LIN {X 0,Y 547.495,Z 446.55,A -85,B 0,C 180,E1 25697.348,E2 25697.348} C_VEL
LIN {X 0,Y 546.646,Z 474.266,A -85,B 0,C 180,E1 25694.031,E2 25694.031} C_VEL
LIN {X 0,Y 545.935,Z 503.573,A -85,B 0,C 180,E1 25690.623,E2 25690.623} C_VEL
LIN {X 0,Y 545.225,Z 533.992,A -85,B 0,C 180,E1 25687.109,E2 25687.109} C_VEL
LIN {X 0,Y 544.841,Z 556.823,A -85,B 0,C 180,E1 25684.577,E2 25684.577} C_VEL
LIN {X 0,Y 545.708,Z 565.508,A -85,B 0,C 180,E1 25684.415,E2 25684.415} C_VEL
LIN {X 0,Y 545.328,Z 668.465,A -85,B 0,C 180,E1 25683.029,E2 25683.029} C_VEL
LIN {X 0,Y 545.205,Z 683.51,A -85,B 0,C 180,E1 25682.627,E2 25682.627} C_VEL
LIN {X 0,Y 545.001,Z 698.163,A -85,B 0,C 180,E1 25682.019,E2 25682.019} C_VEL
LIN {X 0,Y 544.742,Z 711.794,A -85,B 0,C 180,E1 25681.233,E2 25681.233} C_VEL
LIN {X 0,Y 544.518,Z 723.816,A -85,B 0,C 180,E1 25680.329,E2 25680.329} C_VEL
LIN {X 0,Y 544.318,Z 735.754,A -85,B 0,C 180,E1 25679.174,E2 25679.174} C_VEL
LIN {X 0,Y 544.144,Z 746.013,A -85,B 0,C 180,E1 25677.891,E2 25677.891} C_VEL
LIN {X 0,Y 544.028,Z 754.441,A -85,B 0,C 180,E1 25676.526,E2 25676.526} C_VEL
LIN {X 0,Y 543.96,Z 761.021,A -85,B 0,C 180,E1 25675.125,E2 25675.125} C_VEL
LIN {X 0,Y 543.928,Z 766.386,A -85,B 0,C 180,E1 25673.509,E2 25673.509} C_VEL
LIN {X 0,Y 543.917,Z 769.602,A -85,B 0,C 180,E1 25671.911,E2 25671.911} C_VEL
LIN {X 0,Y 543.918,Z 770.918,A -85,B 0,C 180,E1 25670.362,E2 25670.362} C_VEL
LIN {X 0,Y 543.916,Z 770.49,A -85,B 0,C 180,E1 25668.765,E2 25668.765} C_VEL
LIN {X 0,Y 543.919,Z 768.037,A -85,B 0,C 180,E1 25667.105,E2 25667.105} C_VEL
LIN {X 0,Y 543.939,Z 763.873,A -85,B 0,C 180,E1 25665.567,E2 25665.567} C_VEL
LIN {X 0,Y 543.985,Z 758.294,A -85,B 0,C 180,E1 25664.15,E2 25664.15} C_VEL
LIN {X 0,Y 544.074,Z 750.741,A -85,B 0,C 180,E1 25662.74,E2 25662.74} C_VEL
LIN {X 0,Y 544.199,Z 742.577,A -85,B 0,C 180,E1 25661.552,E2 25661.552} C_VEL
LIN {X 0,Y 544.392,Z 731.756,A -85,B 0,C 180,E1 25660.316,E2 25660.316} C_VEL
LIN {X 0,Y 544.604,Z 719.668,A -85,B 0,C 180,E1 25659.244,E2 25659.244} C_VEL
LIN {X 0,Y 544.841,Z 707.24,A -85,B 0,C 180,E1 25658.389,E2 25658.389} C_VEL
LIN {X 0,Y 545.065,Z 694.016,A -85,B 0,C 180,E1 25657.695,E2 25657.695} C_VEL
LIN {X 0,Y 545.26,Z 679.155,A -85,B 0,C 180,E1 25657.146,E2 25657.146} C_VEL
LIN {X 0,Y 545.39,Z 664.539,A -85,B 0,C 180,E1 25656.811,E2 25656.811} C_VEL
LIN {X 0,Y 545.478,Z 561.409,A -85,B 0,C 180,E1 25655.434,E2 25655.434} C_VEL
LIN {X 0,Y 544.883,Z 556.572,A -85,B 0,C 180,E1 25655.317,E2 25655.317} C_VEL
LIN {X 0,Y 545.301,Z 528.031,A -85,B 0,C 180,E1 25652.122,E2 25652.122} C_VEL
LIN {X 0,Y 546.018,Z 497.792,A -85,B 0,C 180,E1 25648.636,E2 25648.636} C_VEL
LIN {X 0,Y 546.669,Z 469.731,A -85,B 0,C 180,E1 25645.384,E2 25645.384} C_VEL
LIN {X 0,Y 547.326,Z 446.384,A -85,B 0,C 180,E1 25642.6,E2 25642.6} C_VEL
LIN {X 0,Y 544.355,Z 435.109,A -85,B 0,C 180,E1 25640.991,E2 25640.991} C_VEL
LIN {X 0,Y 544.39,Z 434.987,A -85,B 0,C 180,E1 25637.806,E2 25637.806} C_VEL
LIN {X 0,Y 544.328,Z 434.99,A -85,B 0,C 180,E1 25634.553,E2 25634.553} C_VEL
LIN {X 0,Y 544.383,Z 434.988,A -85,B 0,C 180,E1 25631.362,E2 25631.362} C_VEL
LIN {X 0,Y 544.329,Z 434.988,A -85,B 0,C 180,E1 25628.22,E2 25628.22} C_VEL
LIN {X 0,Y 544.332,Z 434.989,A -85,B 0,C 180,E1 25624.776,E2 25624.776} C_VEL
LIN {X 0,Y 544.365,Z 434.988,A -85,B 0,C 180,E1 25621.619,E2 25621.619} C_VEL
LIN {X 0,Y 544.318,Z 434.988,A -85,B 0,C 180,E1 25618.431,E2 25618.431} C_VEL
LIN {X 0,Y 544.386,Z 434.991,A -85,B 0,C 180,E1 25615.294,E2 25615.294} C_VEL
LIN {X 0,Y 544.32,Z 434.987,A -85,B 0,C 180,E1 25612.155,E2 25612.155} C_VEL
LIN {X 0,Y 544.373,Z 434.983,A -85,B 0,C 180,E1 25608.887,E2 25608.887} C_VEL
LIN {X 0,Y 544.336,Z 434.987,A -85,B 0,C 180,E1 25605.733,E2 25605.733} C_VEL
LIN {X 0,Y 544.34,Z 434.982,A -85,B 0,C 180,E1 25602.386,E2 25602.386} C_VEL
LIN {X 0,Y 544.365,Z 434.986,A -85,B 0,C 180,E1 25599.322,E2 25599.322} C_VEL
LIN {X 0,Y 544.333,Z 434.985,A -85,B 0,C 180,E1 25596.001,E2 25596.001} C_VEL
LIN {X 0,Y 544.4,Z 434.984,A -85,B 0,C 180,E1 25592.735,E2 25592.735} C_VEL
LIN {X 0,Y 544.34,Z 434.987,A -85,B 0,C 180,E1 25589.611,E2 25589.611} C_VEL
LIN {X 0,Y 544.365,Z 434.976,A -85,B 0,C 180,E1 25586.274,E2 25586.274} C_VEL
LIN {X 0,Y 544.375,Z 434.986,A -85,B 0,C 180,E1 25583.031,E2 25583.031} C_VEL
LIN {X 0,Y 544.346,Z 434.983,A -85,B 0,C 180,E1 25579.754,E2 25579.754} C_VEL
LIN {X 0,Y 544.404,Z 434.98,A -85,B 0,C 180,E1 25576.43,E2 25576.43} C_VEL
LIN {X 0,Y 544.357,Z 434.987,A -85,B 0,C 180,E1 25573.165,E2 25573.165} C_VEL
LIN {X 0,Y 544.359,Z 434.976,A -85,B 0,C 180,E1 25569.729,E2 25569.729} C_VEL
LIN {X 0,Y 544.405,Z 434.985,A -85,B 0,C 180,E1 25566.433,E2 25566.433} C_VEL
LIN {X 0,Y 544.356,Z 434.985,A -85,B 0,C 180,E1 25563.159,E2 25563.159} C_VEL
LIN {X 0,Y 544.382,Z 434.974,A -85,B 0,C 180,E1 25559.79,E2 25559.79} C_VEL
LIN {X 0,Y 544.399,Z 434.989,A -85,B 0,C 180,E1 25556.42,E2 25556.42} C_VEL
LIN {X 0,Y 544.36,Z 434.98,A -85,B 0,C 180,E1 25553.143,E2 25553.143} C_VEL
LIN {X 0,Y 544.402,Z 434.981,A -85,B 0,C 180,E1 25549.845,E2 25549.845} C_VEL
LIN {X 0,Y 544.385,Z 434.987,A -85,B 0,C 180,E1 25546.511,E2 25546.511} C_VEL
LIN {X 0,Y 544.37,Z 434.981,A -85,B 0,C 180,E1 25543.125,E2 25543.125} C_VEL
LIN {X 0,Y 544.401,Z 434.979,A -85,B 0,C 180,E1 25539.801,E2 25539.801} C_VEL
LIN {X 0,Y 544.383,Z 434.985,A -85,B 0,C 180,E1 25536.421,E2 25536.421} C_VEL
LIN {X 0,Y 544.376,Z 434.977,A -85,B 0,C 180,E1 25532.975,E2 25532.975} C_VEL
LIN {X 0,Y 544.4,Z 434.981,A -85,B 0,C 180,E1 25529.664,E2 25529.664} C_VEL
LIN {X 0,Y 544.385,Z 434.986,A -85,B 0,C 180,E1 25526.307,E2 25526.307} C_VEL
LIN {X 0,Y 544.382,Z 434.982,A -85,B 0,C 180,E1 25522.824,E2 25522.824} C_VEL
LIN {X 0,Y 544.396,Z 434.984,A -85,B 0,C 180,E1 25519.446,E2 25519.446} C_VEL
LIN {X 0,Y 544.394,Z 434.988,A -85,B 0,C 180,E1 25516.032,E2 25516.032} C_VEL
LIN {X 0,Y 544.384,Z 434.983,A -85,B 0,C 180,E1 25512.565,E2 25512.565} C_VEL
LIN {X 0,Y 544.393,Z 434.986,A -85,B 0,C 180,E1 25509.32,E2 25509.32} C_VEL
LIN {X 0,Y 544.389,Z 434.986,A -85,B 0,C 180,E1 25505.996,E2 25505.996} C_VEL
LIN {X 0,Y 544.429,Z 435.199,A -85,B 0,C 180,E1 25502.883,E2 25502.883} C_VEL
LIN {X 0,Y 549.545,Z 450.788,A -85,B 0,C 180,E1 25501.295,E2 25501.295} C_VEL
LIN {X 0,Y 548.617,Z 495.169,A -85,B 0,C 180,E1 25498.048,E2 25498.048} C_VEL
LIN {X 0,Y 547.868,Z 539.196,A -85,B 0,C 180,E1 25494.93,E2 25494.93} C_VEL
LIN {X 0,Y 549.12,Z 548.98,A -85,B 0,C 180,E1 25494.728,E2 25494.728} C_VEL
LIN {X 0,Y 548,Z 748.309,A -85,B 0,C 180,E1 25491.965,E2 25491.965} C_VEL
LIN {X 0,Y 547.672,Z 767.397,A -85,B 0,C 180,E1 25491.502,E2 25491.502} C_VEL
LIN {X 0,Y 547.282,Z 785.391,A -85,B 0,C 180,E1 25490.871,E2 25490.871} C_VEL
LIN {X 0,Y 546.836,Z 803.036,A -85,B 0,C 180,E1 25490.05,E2 25490.05} C_VEL
LIN {X 0,Y 546.334,Z 819.765,A -85,B 0,C 180,E1 25489.067,E2 25489.067} C_VEL
LIN {X 0,Y 545.853,Z 835.621,A -85,B 0,C 180,E1 25487.923,E2 25487.923} C_VEL
LIN {X 0,Y 545.378,Z 850.553,A -85,B 0,C 180,E1 25486.619,E2 25486.619} C_VEL
LIN {X 0,Y 544.96,Z 864.211,A -85,B 0,C 180,E1 25485.188,E2 25485.188} C_VEL
LIN {X 0,Y 544.601,Z 876.913,A -85,B 0,C 180,E1 25483.592,E2 25483.592} C_VEL
LIN {X 0,Y 544.329,Z 888.228,A -85,B 0,C 180,E1 25481.872,E2 25481.872} C_VEL
LIN {X 0,Y 544.13,Z 897.993,A -85,B 0,C 180,E1 25480.054,E2 25480.054} C_VEL
LIN {X 0,Y 544.008,Z 906.176,A -85,B 0,C 180,E1 25478.136,E2 25478.136} C_VEL
LIN {X 0,Y 543.945,Z 912.412,A -85,B 0,C 180,E1 25476.226,E2 25476.226} C_VEL
LIN {X 0,Y 543.921,Z 916.878,A -85,B 0,C 180,E1 25474.323,E2 25474.323} C_VEL
LIN {X 0,Y 543.914,Z 919.793,A -85,B 0,C 180,E1 25472.318,E2 25472.318} C_VEL
LIN {X 0,Y 543.908,Z 920.94,A -85,B 0,C 180,E1 25470.316,E2 25470.316} C_VEL
LIN {X 0,Y 543.913,Z 920.347,A -85,B 0,C 180,E1 25468.315,E2 25468.315} C_VEL
LIN {X 0,Y 543.915,Z 918.002,A -85,B 0,C 180,E1 25466.311,E2 25466.311} C_VEL
LIN {X 0,Y 543.931,Z 914.097,A -85,B 0,C 180,E1 25464.409,E2 25464.409} C_VEL
LIN {X 0,Y 543.981,Z 908.468,A -85,B 0,C 180,E1 25462.502,E2 25462.502} C_VEL
LIN {X 0,Y 544.074,Z 901.428,A -85,B 0,C 180,E1 25460.693,E2 25460.693} C_VEL
LIN {X 0,Y 544.234,Z 892.518,A -85,B 0,C 180,E1 25458.878,E2 25458.878} C_VEL
LIN {X 0,Y 544.472,Z 882.154,A -85,B 0,C 180,E1 25457.162,E2 25457.162} C_VEL
LIN {X 0,Y 544.779,Z 870.352,A -85,B 0,C 180,E1 25455.546,E2 25455.546} C_VEL
LIN {X 0,Y 545.178,Z 857.081,A -85,B 0,C 180,E1 25454.032,E2 25454.032} C_VEL
LIN {X 0,Y 545.65,Z 842.222,A -85,B 0,C 180,E1 25452.622,E2 25452.622} C_VEL
LIN {X 0,Y 546.157,Z 826.235,A -85,B 0,C 180,E1 25451.37,E2 25451.37} C_VEL
LIN {X 0,Y 546.65,Z 809.054,A -85,B 0,C 180,E1 25450.278,E2 25450.278} C_VEL
LIN {X 0,Y 547.127,Z 791.811,A -85,B 0,C 180,E1 25449.403,E2 25449.403} C_VEL
LIN {X 0,Y 547.538,Z 773.536,A -85,B 0,C 180,E1 25448.691,E2 25448.691} C_VEL
LIN {X 0,Y 547.894,Z 754.924,A -85,B 0,C 180,E1 25448.174,E2 25448.174} C_VEL
LIN {X 0,Y 548.116,Z 734.498,A -85,B 0,C 180,E1 25447.82,E2 25447.82} C_VEL
LIN {X 0,Y 548.952,Z 546.145,A -85,B 0,C 180,E1 25445.224,E2 25445.224} C_VEL
LIN {X 0,Y 547.799,Z 538.331,A -85,B 0,C 180,E1 25445.034,E2 25445.034} C_VEL
LIN {X 0,Y 548.663,Z 492.747,A -85,B 0,C 180,E1 25441.777,E2 25441.777} C_VEL
LIN {X 0,Y 549.55,Z 450.377,A -85,B 0,C 180,E1 25438.675,E2 25438.675} C_VEL
LIN {X 0,Y 544.437,Z 435.251,A -85,B 0,C 180,E1 25437.134,E2 25437.134} C_VEL
LIN {X 0,Y 544.389,Z 434.988,A -85,B 0,C 180,E1 25433.874,E2 25433.874} C_VEL
LIN {X 0,Y 544.392,Z 434.986,A -85,B 0,C 180,E1 25430.479,E2 25430.479} C_VEL
LIN {X 0,Y 544.4,Z 434.978,A -85,B 0,C 180,E1 25427.048,E2 25427.048} C_VEL
LIN {X 0,Y 544.388,Z 434.986,A -85,B 0,C 180,E1 25423.644,E2 25423.644} C_VEL
LIN {X 0,Y 544.394,Z 434.986,A -85,B 0,C 180,E1 25420.278,E2 25420.278} C_VEL
LIN {X 0,Y 544.4,Z 434.98,A -85,B 0,C 180,E1 25416.911,E2 25416.911} C_VEL
LIN {X 0,Y 544.386,Z 434.984,A -85,B 0,C 180,E1 25413.436,E2 25413.436} C_VEL
LIN {X 0,Y 544.393,Z 434.985,A -85,B 0,C 180,E1 25410.093,E2 25410.093} C_VEL
LIN {X 0,Y 544.395,Z 434.98,A -85,B 0,C 180,E1 25406.742,E2 25406.742} C_VEL
LIN {X 0,Y 544.387,Z 434.985,A -85,B 0,C 180,E1 25403.259,E2 25403.259} C_VEL
LIN {X 0,Y 544.394,Z 434.984,A -85,B 0,C 180,E1 25399.888,E2 25399.888} C_VEL
LIN {X 0,Y 544.4,Z 434.979,A -85,B 0,C 180,E1 25396.43,E2 25396.43} C_VEL
LIN {X 0,Y 544.385,Z 434.986,A -85,B 0,C 180,E1 25393.056,E2 25393.056} C_VEL
LIN {X 0,Y 544.393,Z 434.981,A -85,B 0,C 180,E1 25389.728,E2 25389.728} C_VEL
LIN {X 0,Y 544.393,Z 434.98,A -85,B 0,C 180,E1 25386.327,E2 25386.327} C_VEL
LIN {X 0,Y 544.384,Z 434.986,A -85,B 0,C 180,E1 25382.842,E2 25382.842} C_VEL
LIN {X 0,Y 544.395,Z 434.98,A -85,B 0,C 180,E1 25379.474,E2 25379.474} C_VEL
LIN {X 0,Y 544.392,Z 434.979,A -85,B 0,C 180,E1 25376.103,E2 25376.103} C_VEL
LIN {X 0,Y 544.385,Z 434.986,A -85,B 0,C 180,E1 25372.659,E2 25372.659} C_VEL
LIN {X 0,Y 544.395,Z 434.98,A -85,B 0,C 180,E1 25369.296,E2 25369.296} C_VEL
LIN {X 0,Y 544.393,Z 434.977,A -85,B 0,C 180,E1 25365.871,E2 25365.871} C_VEL
LIN {X 0,Y 544.381,Z 434.984,A -85,B 0,C 180,E1 25362.409,E2 25362.409} C_VEL
LIN {X 0,Y 544.397,Z 434.985,A -85,B 0,C 180,E1 25359.013,E2 25359.013} C_VEL
LIN {X 0,Y 544.395,Z 434.977,A -85,B 0,C 180,E1 25355.591,E2 25355.591} C_VEL
LIN {X 0,Y 544.382,Z 434.987,A -85,B 0,C 180,E1 25352.191,E2 25352.191} C_VEL
LIN {X 0,Y 544.4,Z 434.982,A -85,B 0,C 180,E1 25349.102,E2 25349.102} C_VEL
LIN {X 0,Y 543.39,Z 435.113,A -85,B 0,C 180,E1 25348.291,E2 25348.291} C_VEL
LIN {X 0,Y 536.961,Z 435.911,A -85,B 0,C 180,E1 25346.014,E2 25346.014} C_VEL
LIN {X 0,Y 536.452,Z 435.971,A -85,B 0,C 180,E1 25345.421,E2 25345.421} C_VEL
LIN {X 0,Y 536.445,Z 435.977,A -85,B 0,C 180,E1 25342.037,E2 25342.037} C_VEL
LIN {X 0,Y 536.485,Z 436.227,A -85,B 0,C 180,E1 25339.335,E2 25339.335} C_VEL
LIN {X 0,Y 539.968,Z 449.754,A -85,B 0,C 180,E1 25337.406,E2 25337.406} C_VEL
LIN {X 0,Y 538.979,Z 478.583,A -85,B 0,C 180,E1 25333.932,E2 25333.932} C_VEL
LIN {X 0,Y 538.235,Z 506.906,A -85,B 0,C 180,E1 25330.6,E2 25330.6} C_VEL
LIN {X 0,Y 537.432,Z 537.08,A -85,B 0,C 180,E1 25327.069,E2 25327.069} C_VEL
LIN {X 0,Y 537.047,Z 556.841,A -85,B 0,C 180,E1 25324.835,E2 25324.835} C_VEL
LIN {X 0,Y 538.032,Z 566.096,A -85,B 0,C 180,E1 25324.647,E2 25324.647} C_VEL
LIN {X 0,Y 537.537,Z 668.696,A -85,B 0,C 180,E1 25323.219,E2 25323.219} C_VEL
LIN {X 0,Y 537.393,Z 683.257,A -85,B 0,C 180,E1 25322.823,E2 25322.823} C_VEL
LIN {X 0,Y 537.162,Z 698.051,A -85,B 0,C 180,E1 25322.203,E2 25322.203} C_VEL
LIN {X 0,Y 536.879,Z 711.35,A -85,B 0,C 180,E1 25321.43,E2 25321.43} C_VEL
LIN {X 0,Y 536.617,Z 723.478,A -85,B 0,C 180,E1 25320.513,E2 25320.513} C_VEL
LIN {X 0,Y 536.389,Z 735.343,A -85,B 0,C 180,E1 25319.357,E2 25319.357} C_VEL
LIN {X 0,Y 536.194,Z 745.279,A -85,B 0,C 180,E1 25318.112,E2 25318.112} C_VEL
LIN {X 0,Y 536.062,Z 753.333,A -85,B 0,C 180,E1 25316.832,E2 25316.832} C_VEL
LIN {X 0,Y 535.971,Z 760.681,A -85,B 0,C 180,E1 25315.29,E2 25315.29} C_VEL
LIN {X 0,Y 535.932,Z 765.819,A -85,B 0,C 180,E1 25313.764,E2 25313.764} C_VEL
LIN {X 0,Y 535.919,Z 769.129,A -85,B 0,C 180,E1 25312.255,E2 25312.255} C_VEL
LIN {X 0,Y 535.918,Z 770.822,A -85,B 0,C 180,E1 25310.647,E2 25310.647} C_VEL
LIN {X 0,Y 535.916,Z 770.693,A -85,B 0,C 180,E1 25309.056,E2 25309.056} C_VEL
LIN {X 0,Y 535.919,Z 768.842,A -85,B 0,C 180,E1 25307.48,E2 25307.48} C_VEL
LIN {X 0,Y 535.937,Z 764.857,A -85,B 0,C 180,E1 25305.806,E2 25305.806} C_VEL
LIN {X 0,Y 535.987,Z 759.124,A -85,B 0,C 180,E1 25304.255,E2 25304.255} C_VEL
LIN {X 0,Y 536.082,Z 751.872,A -85,B 0,C 180,E1 25302.823,E2 25302.823} C_VEL
LIN {X 0,Y 536.233,Z 743.203,A -85,B 0,C 180,E1 25301.508,E2 25301.508} C_VEL
LIN {X 0,Y 536.453,Z 732.279,A -85,B 0,C 180,E1 25300.227,E2 25300.227} C_VEL
LIN {X 0,Y 536.689,Z 720.664,A -85,B 0,C 180,E1 25299.165,E2 25299.165} C_VEL
LIN {X 0,Y 536.953,Z 708.57,A -85,B 0,C 180,E1 25298.297,E2 25298.297} C_VEL
LIN {X 0,Y 537.22,Z 694.554,A -85,B 0,C 180,E1 25297.539,E2 25297.539} C_VEL
LIN {X 0,Y 537.436,Z 680.185,A -85,B 0,C 180,E1 25296.989,E2 25296.989} C_VEL
LIN {X 0,Y 537.598,Z 665.309,A -85,B 0,C 180,E1 25296.628,E2 25296.628} C_VEL
LIN {X 0,Y 537.808,Z 562.279,A -85,B 0,C 180,E1 25295.207,E2 25295.207} C_VEL
LIN {X 0,Y 537.071,Z 556.649,A -85,B 0,C 180,E1 25295.073,E2 25295.073} C_VEL
LIN {X 0,Y 537.587,Z 528.08,A -85,B 0,C 180,E1 25291.812,E2 25291.812} C_VEL
LIN {X 0,Y 538.382,Z 497.987,A -85,B 0,C 180,E1 25288.297,E2 25288.297} C_VEL
LIN {X 0,Y 539.146,Z 469.958,A -85,B 0,C 180,E1 25284.999,E2 25284.999} C_VEL
LIN {X 0,Y 539.763,Z 448.718,A -85,B 0,C 180,E1 25282.442,E2 25282.442} C_VEL
LIN {X 0,Y 536.412,Z 436.103,A -85,B 0,C 180,E1 25280.613,E2 25280.613} C_VEL
LIN {X 0,Y 536.428,Z 435.978,A -85,B 0,C 180,E1 25277.294,E2 25277.294} C_VEL
LIN {X 0,Y 536.402,Z 435.978,A -85,B 0,C 180,E1 25274.208,E2 25274.208} C_VEL
LIN {X 0,Y 536.391,Z 435.977,A -85,B 0,C 180,E1 25270.735,E2 25270.735} C_VEL
LIN {X 0,Y 536.455,Z 435.965,A -85,B 0,C 180,E1 25267.537,E2 25267.537} C_VEL
LIN {X 0,Y 536.384,Z 435.978,A -85,B 0,C 180,E1 25264.257,E2 25264.257} C_VEL
LIN {X 0,Y 536.404,Z 435.979,A -85,B 0,C 180,E1 25260.889,E2 25260.889} C_VEL
LIN {X 0,Y 536.399,Z 435.976,A -85,B 0,C 180,E1 25257.784,E2 25257.784} C_VEL
LIN {X 0,Y 536.384,Z 435.977,A -85,B 0,C 180,E1 25254.437,E2 25254.437} C_VEL
LIN {X 0,Y 536.456,Z 435.977,A -85,B 0,C 180,E1 25251.177,E2 25251.177} C_VEL
LIN {X 0,Y 536.387,Z 435.973,A -85,B 0,C 180,E1 25247.994,E2 25247.994} C_VEL
LIN {X 0,Y 536.419,Z 435.976,A -85,B 0,C 180,E1 25244.645,E2 25244.645} C_VEL
LIN {X 0,Y 536.413,Z 435.972,A -85,B 0,C 180,E1 25241.468,E2 25241.468} C_VEL
LIN {X 0,Y 536.395,Z 435.977,A -85,B 0,C 180,E1 25238.097,E2 25238.097} C_VEL
LIN {X 0,Y 536.458,Z 435.966,A -85,B 0,C 180,E1 25234.904,E2 25234.904} C_VEL
LIN {X 0,Y 536.399,Z 435.975,A -85,B 0,C 180,E1 25231.713,E2 25231.713} C_VEL
LIN {X 0,Y 536.432,Z 435.97,A -85,B 0,C 180,E1 25228.379,E2 25228.379} C_VEL
LIN {X 0,Y 536.426,Z 435.967,A -85,B 0,C 180,E1 25225.149,E2 25225.149} C_VEL
LIN {X 0,Y 536.407,Z 435.975,A -85,B 0,C 180,E1 25221.774,E2 25221.774} C_VEL
LIN {X 0,Y 536.461,Z 435.961,A -85,B 0,C 180,E1 25218.473,E2 25218.473} C_VEL
LIN {X 0,Y 536.414,Z 435.972,A -85,B 0,C 180,E1 25215.238,E2 25215.238} C_VEL
LIN {X 0,Y 536.417,Z 435.972,A -85,B 0,C 180,E1 25211.723,E2 25211.723} C_VEL
LIN {X 0,Y 536.465,Z 435.964,A -85,B 0,C 180,E1 25208.467,E2 25208.467} C_VEL
LIN {X 0,Y 536.419,Z 435.974,A -85,B 0,C 180,E1 25205.133,E2 25205.133} C_VEL
LIN {X 0,Y 536.432,Z 435.966,A -85,B 0,C 180,E1 25201.709,E2 25201.709} C_VEL
LIN {X 0,Y 536.465,Z 435.97,A -85,B 0,C 180,E1 25198.398,E2 25198.398} C_VEL
LIN {X 0,Y 536.421,Z 435.974,A -85,B 0,C 180,E1 25195.082,E2 25195.082} C_VEL
LIN {X 0,Y 536.457,Z 435.963,A -85,B 0,C 180,E1 25191.749,E2 25191.749} C_VEL
LIN {X 0,Y 536.457,Z 435.977,A -85,B 0,C 180,E1 25188.388,E2 25188.388} C_VEL
LIN {X 0,Y 536.425,Z 435.966,A -85,B 0,C 180,E1 25184.984,E2 25184.984} C_VEL
LIN {X 0,Y 536.462,Z 435.97,A -85,B 0,C 180,E1 25181.64,E2 25181.64} C_VEL
LIN {X 0,Y 536.463,Z 435.97,A -85,B 0,C 180,E1 25178.152,E2 25178.152} C_VEL
LIN {X 0,Y 536.434,Z 435.973,A -85,B 0,C 180,E1 25174.733,E2 25174.733} C_VEL
LIN {X 0,Y 536.467,Z 435.969,A -85,B 0,C 180,E1 25171.381,E2 25171.381} C_VEL
LIN {X 0,Y 536.464,Z 435.972,A -85,B 0,C 180,E1 25167.915,E2 25167.915} C_VEL
LIN {X 0,Y 536.438,Z 435.972,A -85,B 0,C 180,E1 25164.54,E2 25164.54} C_VEL
LIN {X 0,Y 536.462,Z 435.967,A -85,B 0,C 180,E1 25161.09,E2 25161.09} C_VEL
LIN {X 0,Y 536.461,Z 435.973,A -85,B 0,C 180,E1 25157.714,E2 25157.714} C_VEL
LIN {X 0,Y 536.444,Z 435.972,A -85,B 0,C 180,E1 25154.298,E2 25154.298} C_VEL
LIN {X 0,Y 536.463,Z 435.971,A -85,B 0,C 180,E1 25150.826,E2 25150.826} C_VEL
LIN {X 0,Y 536.456,Z 435.977,A -85,B 0,C 180,E1 25147.417,E2 25147.417} C_VEL
LIN {X 0,Y 536.451,Z 435.976,A -85,B 0,C 180,E1 25143.997,E2 25143.997} C_VEL
LIN {X 0,Y 536.508,Z 436.346,A -85,B 0,C 180,E1 25143.282,E2 25143.282} C_VEL
LIN {X 0,Y 542.232,Z 453.381,A -85,B 0,C 180,E1 25141.524,E2 25141.524} C_VEL
LIN {X 0,Y 541.159,Z 496.053,A -85,B 0,C 180,E1 25138.349,E2 25138.349} C_VEL
LIN {X 0,Y 540.28,Z 539.241,A -85,B 0,C 180,E1 25135.245,E2 25135.245} C_VEL
LIN {X 0,Y 541.72,Z 550.007,A -85,B 0,C 180,E1 25135.037,E2 25135.037} C_VEL
LIN {X 0,Y 540.616,Z 745.193,A -85,B 0,C 180,E1 25132.336,E2 25132.336} C_VEL
LIN {X 0,Y 540.277,Z 763.946,A -85,B 0,C 180,E1 25131.913,E2 25131.913} C_VEL
LIN {X 0,Y 539.846,Z 781.952,A -85,B 0,C 180,E1 25131.312,E2 25131.312} C_VEL
LIN {X 0,Y 539.37,Z 799.844,A -85,B 0,C 180,E1 25130.51,E2 25130.51} C_VEL
LIN {X 0,Y 538.786,Z 817.24,A -85,B 0,C 180,E1 25129.514,E2 25129.514} C_VEL
LIN {X 0,Y 538.22,Z 833.955,A -85,B 0,C 180,E1 25128.324,E2 25128.324} C_VEL
LIN {X 0,Y 537.655,Z 849.441,A -85,B 0,C 180,E1 25126.976,E2 25126.976} C_VEL
LIN {X 0,Y 537.171,Z 863.091,A -85,B 0,C 180,E1 25125.547,E2 25125.547} C_VEL
LIN {X 0,Y 536.736,Z 876.14,A -85,B 0,C 180,E1 25123.905,E2 25123.905} C_VEL
LIN {X 0,Y 536.408,Z 887.592,A -85,B 0,C 180,E1 25122.16,E2 25122.16} C_VEL
LIN {X 0,Y 536.175,Z 897.478,A -85,B 0,C 180,E1 25120.313,E2 25120.313} C_VEL
LIN {X 0,Y 536.036,Z 905.771,A -85,B 0,C 180,E1 25118.366,E2 25118.366} C_VEL
LIN {X 0,Y 535.953,Z 912.109,A -85,B 0,C 180,E1 25116.427,E2 25116.427} C_VEL
LIN {X 0,Y 535.923,Z 916.877,A -85,B 0,C 180,E1 25114.387,E2 25114.387} C_VEL
LIN {X 0,Y 535.913,Z 919.794,A -85,B 0,C 180,E1 25112.353,E2 25112.353} C_VEL
LIN {X 0,Y 535.908,Z 920.94,A -85,B 0,C 180,E1 25110.321,E2 25110.321} C_VEL
LIN {X 0,Y 535.913,Z 920.346,A -85,B 0,C 180,E1 25108.29,E2 25108.29} C_VEL
LIN {X 0,Y 535.917,Z 918.002,A -85,B 0,C 180,E1 25106.256,E2 25106.256} C_VEL
LIN {X 0,Y 535.935,Z 914.097,A -85,B 0,C 180,E1 25104.326,E2 25104.326} C_VEL
LIN {X 0,Y 535.995,Z 908.468,A -85,B 0,C 180,E1 25102.389,E2 25102.389} C_VEL
LIN {X 0,Y 536.099,Z 901.428,A -85,B 0,C 180,E1 25100.554,E2 25100.554} C_VEL
LIN {X 0,Y 536.287,Z 892.518,A -85,B 0,C 180,E1 25098.711,E2 25098.711} C_VEL
LIN {X 0,Y 536.561,Z 882.154,A -85,B 0,C 180,E1 25096.969,E2 25096.969} C_VEL
LIN {X 0,Y 536.916,Z 870.353,A -85,B 0,C 180,E1 25095.33,E2 25095.33} C_VEL
LIN {X 0,Y 537.392,Z 856.685,A -85,B 0,C 180,E1 25093.751,E2 25093.751} C_VEL
LIN {X 0,Y 537.944,Z 841.605,A -85,B 0,C 180,E1 25092.309,E2 25092.309} C_VEL
LIN {X 0,Y 538.52,Z 825.441,A -85,B 0,C 180,E1 25091.04,E2 25091.04} C_VEL
LIN {X 0,Y 539.071,Z 808.706,A -85,B 0,C 180,E1 25089.969,E2 25089.969} C_VEL
LIN {X 0,Y 539.594,Z 791.813,A -85,B 0,C 180,E1 25089.103,E2 25089.103} C_VEL
LIN {X 0,Y 540.059,Z 773.537,A -85,B 0,C 180,E1 25088.382,E2 25088.382} C_VEL
LIN {X 0,Y 540.46,Z 754.851,A -85,B 0,C 180,E1 25087.856,E2 25087.856} C_VEL
LIN {X 0,Y 540.711,Z 734.244,A -85,B 0,C 180,E1 25087.496,E2 25087.496} C_VEL
LIN {X 0,Y 541.594,Z 547.529,A -85,B 0,C 180,E1 25084.926,E2 25084.926} C_VEL
LIN {X 0,Y 540.213,Z 538.244,A -85,B 0,C 180,E1 25084.715,E2 25084.715} C_VEL
LIN {X 0,Y 541.214,Z 493.631,A -85,B 0,C 180,E1 25081.474,E2 25081.474} C_VEL
LIN {X 0,Y 542.216,Z 452.994,A -85,B 0,C 180,E1 25078.447,E2 25078.447} C_VEL
LIN {X 0,Y 536.484,Z 436.208,A -85,B 0,C 180,E1 25076.695,E2 25076.695} C_VEL
LIN {X 0,Y 536.456,Z 435.972,A -85,B 0,C 180,E1 25073.386,E2 25073.386} C_VEL
LIN {X 0,Y 536.457,Z 435.974,A -85,B 0,C 180,E1 25069.983,E2 25069.983} C_VEL
LIN {X 0,Y 536.452,Z 435.971,A -85,B 0,C 180,E1 25066.548,E2 25066.548} C_VEL
LIN {X 0,Y 536.455,Z 435.971,A -85,B 0,C 180,E1 25063.159,E2 25063.159} C_VEL
LIN {X 0,Y 536.452,Z 435.971,A -85,B 0,C 180,E1 25059.667,E2 25059.667} C_VEL
LIN {X 0,Y 536.453,Z 435.973,A -85,B 0,C 180,E1 25056.349,E2 25056.349} C_VEL
LIN {X 0,Y 536.453,Z 435.968,A -85,B 0,C 180,E1 25052.973,E2 25052.973} C_VEL
LIN {X 0,Y 536.452,Z 435.972,A -85,B 0,C 180,E1 25049.475,E2 25049.475} C_VEL
LIN {X 0,Y 536.454,Z 435.973,A -85,B 0,C 180,E1 25046.056,E2 25046.056} C_VEL
LIN {X 0,Y 536.461,Z 435.968,A -85,B 0,C 180,E1 25042.578,E2 25042.578} C_VEL
LIN {X 0,Y 536.447,Z 435.971,A -85,B 0,C 180,E1 25039.15,E2 25039.15} C_VEL
LIN {X 0,Y 536.457,Z 435.974,A -85,B 0,C 180,E1 25035.79,E2 25035.79} C_VEL
LIN {X 0,Y 536.459,Z 435.969,A -85,B 0,C 180,E1 25032.377,E2 25032.377} C_VEL
LIN {X 0,Y 536.444,Z 435.972,A -85,B 0,C 180,E1 25028.899,E2 25028.899} C_VEL
LIN {X 0,Y 536.456,Z 435.974,A -85,B 0,C 180,E1 25025.562,E2 25025.562} C_VEL
LIN {X 0,Y 536.459,Z 435.969,A -85,B 0,C 180,E1 25022.136,E2 25022.136} C_VEL
LIN {X 0,Y 536.445,Z 435.974,A -85,B 0,C 180,E1 25018.718,E2 25018.718} C_VEL
LIN {X 0,Y 536.458,Z 435.972,A -85,B 0,C 180,E1 25015.296,E2 25015.296} C_VEL
LIN {X 0,Y 536.463,Z 435.968,A -85,B 0,C 180,E1 25011.856,E2 25011.856} C_VEL
LIN {X 0,Y 536.442,Z 435.973,A -85,B 0,C 180,E1 25008.387,E2 25008.387} C_VEL
LIN {X 0,Y 536.461,Z 435.972,A -85,B 0,C 180,E1 25004.985,E2 25004.985} C_VEL
LIN {X 0,Y 536.461,Z 435.967,A -85,B 0,C 180,E1 25001.527,E2 25001.527} C_VEL
LIN {X 0,Y 536.441,Z 435.973,A -85,B 0,C 180,E1 24998.113,E2 24998.113} C_VEL
LIN {X 0,Y 536.462,Z 435.974,A -85,B 0,C 180,E1 24994.681,E2 24994.681} C_VEL
LIN {X 0,Y 536.464,Z 435.97,A -85,B 0,C 180,E1 24991.258,E2 24991.258} C_VEL
LIN {X 0,Y 536.44,Z 435.973,A -85,B 0,C 180,E1 24987.913,E2 24987.913} C_VEL
LIN {X 0,Y 536.452,Z 435.971,A -85,B 0,C 180,E1 24985.421,E2 24985.421} C_VEL
LIN {X 0,Y 535.485,Z 436.099,A -85,B 0,C 180,E1 24984.598,E2 24984.598} C_VEL
LIN {X 0,Y 529.028,Z 436.905,A -85,B 0,C 180,E1 24982.287,E2 24982.287} C_VEL
LIN {X 0,Y 528.5,Z 436.968,A -85,B 0,C 180,E1 24981.685,E2 24981.685} C_VEL
LIN {X 0,Y 528.538,Z 437.24,A -85,B 0,C 180,E1 24979.742,E2 24979.742} C_VEL
LIN {X 0,Y 532.487,Z 451.799,A -85,B 0,C 180,E1 24977.615,E2 24977.615} C_VEL
LIN {X 0,Y 531.412,Z 480.504,A -85,B 0,C 180,E1 24974.12,E2 24974.12} C_VEL
LIN {X 0,Y 530.573,Z 508.777,A -85,B 0,C 180,E1 24970.75,E2 24970.75} C_VEL
LIN {X 0,Y 529.683,Z 538.757,A -85,B 0,C 180,E1 24967.194,E2 24967.194} C_VEL
LIN {X 0,Y 529.316,Z 556.744,A -85,B 0,C 180,E1 24965.144,E2 24965.144} C_VEL
LIN {X 0,Y 530.523,Z 566.885,A -85,B 0,C 180,E1 24964.935,E2 24964.935} C_VEL
LIN {X 0,Y 529.939,Z 669.101,A -85,B 0,C 180,E1 24963.485,E2 24963.485} C_VEL
LIN {X 0,Y 529.767,Z 683.973,A -85,B 0,C 180,E1 24963.071,E2 24963.071} C_VEL
LIN {X 0,Y 529.477,Z 698.928,A -85,B 0,C 180,E1 24962.423,E2 24962.423} C_VEL
LIN {X 0,Y 529.121,Z 712.409,A -85,B 0,C 180,E1 24961.607,E2 24961.607} C_VEL
LIN {X 0,Y 528.799,Z 723.971,A -85,B 0,C 180,E1 24960.698,E2 24960.698} C_VEL
LIN {X 0,Y 528.498,Z 735.707,A -85,B 0,C 180,E1 24959.509,E2 24959.509} C_VEL
LIN {X 0,Y 528.247,Z 745.422,A -85,B 0,C 180,E1 24958.242,E2 24958.242} C_VEL
LIN {X 0,Y 528.07,Z 754.132,A -85,B 0,C 180,E1 24956.784,E2 24956.784} C_VEL
LIN {X 0,Y 527.977,Z 760.805,A -85,B 0,C 180,E1 24955.34,E2 24955.34} C_VEL
LIN {X 0,Y 527.932,Z 766.236,A -85,B 0,C 180,E1 24953.672,E2 24953.672} C_VEL
LIN {X 0,Y 527.92,Z 769.52,A -85,B 0,C 180,E1 24952.024,E2 24952.024} C_VEL
LIN {X 0,Y 527.918,Z 770.889,A -85,B 0,C 180,E1 24950.511,E2 24950.511} C_VEL
LIN {X 0,Y 527.916,Z 770.529,A -85,B 0,C 180,E1 24948.782,E2 24948.782} C_VEL
LIN {X 0,Y 527.92,Z 768.353,A -85,B 0,C 180,E1 24947.185,E2 24947.185} C_VEL
LIN {X 0,Y 527.944,Z 764.413,A -85,B 0,C 180,E1 24945.6,E2 24945.6} C_VEL
LIN {X 0,Y 528.006,Z 758.53,A -85,B 0,C 180,E1 24944.027,E2 24944.027} C_VEL
LIN {X 0,Y 528.122,Z 751.079,A -85,B 0,C 180,E1 24942.575,E2 24942.575} C_VEL
LIN {X 0,Y 528.317,Z 742.372,A -85,B 0,C 180,E1 24941.241,E2 24941.241} C_VEL
LIN {X 0,Y 528.6,Z 731.705,A -85,B 0,C 180,E1 24939.966,E2 24939.966} C_VEL
LIN {X 0,Y 528.91,Z 719.754,A -85,B 0,C 180,E1 24938.863,E2 24938.863} C_VEL
LIN {X 0,Y 529.247,Z 707.404,A -85,B 0,C 180,E1 24937.982,E2 24937.982} C_VEL
LIN {X 0,Y 529.554,Z 694.276,A -85,B 0,C 180,E1 24937.267,E2 24937.267} C_VEL
LIN {X 0,Y 529.822,Z 679.157,A -85,B 0,C 180,E1 24936.692,E2 24936.692} C_VEL
LIN {X 0,Y 529.986,Z 664.36,A -85,B 0,C 180,E1 24936.348,E2 24936.348} C_VEL
LIN {X 0,Y 530.273,Z 563.237,A -85,B 0,C 180,E1 24934.932,E2 24934.932} C_VEL
LIN {X 0,Y 529.301,Z 556.43,A -85,B 0,C 180,E1 24934.768,E2 24934.768} C_VEL
LIN {X 0,Y 529.885,Z 528.312,A -85,B 0,C 180,E1 24931.514,E2 24931.514} C_VEL
LIN {X 0,Y 530.743,Z 499.095,A -85,B 0,C 180,E1 24928.057,E2 24928.057} C_VEL
LIN {X 0,Y 531.614,Z 471.08,A -85,B 0,C 180,E1 24924.712,E2 24924.712} C_VEL
LIN {X 0,Y 532.328,Z 451.582,A -85,B 0,C 180,E1 24922.336,E2 24922.336} C_VEL
LIN {X 0,Y 528.488,Z 437.083,A -85,B 0,C 180,E1 24920.226,E2 24920.226} C_VEL
LIN {X 0,Y 528.457,Z 436.968,A -85,B 0,C 180,E1 24916.877,E2 24916.877} C_VEL
LIN {X 0,Y 528.518,Z 436.966,A -85,B 0,C 180,E1 24913.627,E2 24913.627} C_VEL
LIN {X 0,Y 528.451,Z 436.966,A -85,B 0,C 180,E1 24910.319,E2 24910.319} C_VEL
LIN {X 0,Y 528.458,Z 436.952,A -85,B 0,C 180,E1 24906.858,E2 24906.858} C_VEL
LIN {X 0,Y 528.495,Z 436.966,A -85,B 0,C 180,E1 24903.602,E2 24903.602} C_VEL
LIN {X 0,Y 528.442,Z 436.968,A -85,B 0,C 180,E1 24900.407,E2 24900.407} C_VEL
LIN {X 0,Y 528.498,Z 436.965,A -85,B 0,C 180,E1 24897.114,E2 24897.114} C_VEL
LIN {X 0,Y 528.456,Z 436.966,A -85,B 0,C 180,E1 24893.82,E2 24893.82} C_VEL
LIN {X 0,Y 528.449,Z 436.967,A -85,B 0,C 180,E1 24890.361,E2 24890.361} C_VEL
LIN {X 0,Y 528.515,Z 436.96,A -85,B 0,C 180,E1 24887.073,E2 24887.073} C_VEL
LIN {X 0,Y 528.453,Z 436.967,A -85,B 0,C 180,E1 24883.828,E2 24883.828} C_VEL
LIN {X 0,Y 528.473,Z 436.961,A -85,B 0,C 180,E1 24880.463,E2 24880.463} C_VEL
LIN {X 0,Y 528.479,Z 436.967,A -85,B 0,C 180,E1 24877.38,E2 24877.38} C_VEL
LIN {X 0,Y 528.459,Z 436.954,A -85,B 0,C 180,E1 24874.033,E2 24874.033} C_VEL
LIN {X 0,Y 528.527,Z 436.963,A -85,B 0,C 180,E1 24870.716,E2 24870.716} C_VEL
LIN {X 0,Y 528.473,Z 436.961,A -85,B 0,C 180,E1 24867.371,E2 24867.371} C_VEL
LIN {X 0,Y 528.468,Z 436.961,A -85,B 0,C 180,E1 24863.884,E2 24863.884} C_VEL
LIN {X 0,Y 528.528,Z 436.96,A -85,B 0,C 180,E1 24860.602,E2 24860.602} C_VEL
LIN {X 0,Y 528.473,Z 436.951,A -85,B 0,C 180,E1 24857.28,E2 24857.28} C_VEL
LIN {X 0,Y 528.479,Z 436.962,A -85,B 0,C 180,E1 24853.792,E2 24853.792} C_VEL
LIN {X 0,Y 528.527,Z 436.954,A -85,B 0,C 180,E1 24850.464,E2 24850.464} C_VEL
LIN {X 0,Y 528.478,Z 436.956,A -85,B 0,C 180,E1 24847.173,E2 24847.173} C_VEL
LIN {X 0,Y 528.489,Z 436.96,A -85,B 0,C 180,E1 24843.688,E2 24843.688} C_VEL
LIN {X 0,Y 528.527,Z 436.951,A -85,B 0,C 180,E1 24840.325,E2 24840.325} C_VEL
LIN {X 0,Y 528.485,Z 436.963,A -85,B 0,C 180,E1 24836.964,E2 24836.964} C_VEL
LIN {X 0,Y 528.493,Z 436.956,A -85,B 0,C 180,E1 24833.482,E2 24833.482} C_VEL
LIN {X 0,Y 528.526,Z 436.962,A -85,B 0,C 180,E1 24830.087,E2 24830.087} C_VEL
LIN {X 0,Y 528.493,Z 436.963,A -85,B 0,C 180,E1 24826.767,E2 24826.767} C_VEL
LIN {X 0,Y 528.499,Z 436.957,A -85,B 0,C 180,E1 24823.288,E2 24823.288} C_VEL
LIN {X 0,Y 528.524,Z 436.957,A -85,B 0,C 180,E1 24819.861,E2 24819.861} C_VEL
LIN {X 0,Y 528.502,Z 436.962,A -85,B 0,C 180,E1 24816.473,E2 24816.473} C_VEL
LIN {X 0,Y 528.5,Z 436.954,A -85,B 0,C 180,E1 24812.996,E2 24812.996} C_VEL
LIN {X 0,Y 528.523,Z 436.958,A -85,B 0,C 180,E1 24809.617,E2 24809.617} C_VEL
LIN {X 0,Y 528.516,Z 436.965,A -85,B 0,C 180,E1 24806.152,E2 24806.152} C_VEL
LIN {X 0,Y 528.502,Z 436.961,A -85,B 0,C 180,E1 24802.743,E2 24802.743} C_VEL
LIN {X 0,Y 528.521,Z 436.961,A -85,B 0,C 180,E1 24799.343,E2 24799.343} C_VEL
LIN {X 0,Y 528.524,Z 436.965,A -85,B 0,C 180,E1 24795.807,E2 24795.807} C_VEL
LIN {X 0,Y 528.505,Z 436.964,A -85,B 0,C 180,E1 24792.338,E2 24792.338} C_VEL
LIN {X 0,Y 528.525,Z 436.961,A -85,B 0,C 180,E1 24788.908,E2 24788.908} C_VEL
LIN {X 0,Y 528.517,Z 436.966,A -85,B 0,C 180,E1 24785.376,E2 24785.376} C_VEL
LIN {X 0,Y 528.561,Z 437.255,A -85,B 0,C 180,E1 24783.741,E2 24783.741} C_VEL
LIN {X 0,Y 534.914,Z 456.279,A -85,B 0,C 180,E1 24781.736,E2 24781.736} C_VEL
LIN {X 0,Y 533.782,Z 494.51,A -85,B 0,C 180,E1 24778.838,E2 24778.838} C_VEL
LIN {X 0,Y 532.664,Z 536.717,A -85,B 0,C 180,E1 24775.71,E2 24775.71} C_VEL
LIN {X 0,Y 532.709,Z 539.722,A -85,B 0,C 180,E1 24775.536,E2 24775.536} C_VEL
LIN {X 0,Y 534.201,Z 550.976,A -85,B 0,C 180,E1 24775.318,E2 24775.318} C_VEL
LIN {X 0,Y 533.105,Z 748.238,A -85,B 0,C 180,E1 24772.59,E2 24772.59} C_VEL
LIN {X 0,Y 532.735,Z 767.551,A -85,B 0,C 180,E1 24772.121,E2 24772.121} C_VEL
LIN {X 0,Y 532.27,Z 785.383,A -85,B 0,C 180,E1 24771.488,E2 24771.488} C_VEL
LIN {X 0,Y 531.706,Z 803.03,A -85,B 0,C 180,E1 24770.646,E2 24770.646} C_VEL
LIN {X 0,Y 531.068,Z 819.759,A -85,B 0,C 180,E1 24769.638,E2 24769.638} C_VEL
LIN {X 0,Y 530.456,Z 835.616,A -85,B 0,C 180,E1 24768.462,E2 24768.462} C_VEL
LIN {X 0,Y 529.847,Z 850.55,A -85,B 0,C 180,E1 24767.121,E2 24767.121} C_VEL
LIN {X 0,Y 529.309,Z 864.017,A -85,B 0,C 180,E1 24765.672,E2 24765.672} C_VEL
LIN {X 0,Y 528.854,Z 876.275,A -85,B 0,C 180,E1 24764.097,E2 24764.097} C_VEL
LIN {X 0,Y 528.482,Z 887.591,A -85,B 0,C 180,E1 24762.345,E2 24762.345} C_VEL
LIN {X 0,Y 528.217,Z 897.477,A -85,B 0,C 180,E1 24760.47,E2 24760.47} C_VEL
LIN {X 0,Y 528.052,Z 905.771,A -85,B 0,C 180,E1 24758.493,E2 24758.493} C_VEL
LIN {X 0,Y 527.96,Z 912.109,A -85,B 0,C 180,E1 24756.525,E2 24756.525} C_VEL
LIN {X 0,Y 527.924,Z 916.877,A -85,B 0,C 180,E1 24754.454,E2 24754.454} C_VEL
LIN {X 0,Y 527.912,Z 919.793,A -85,B 0,C 180,E1 24752.388,E2 24752.388} C_VEL
LIN {X 0,Y 527.908,Z 920.939,A -85,B 0,C 180,E1 24750.326,E2 24750.326} C_VEL
LIN {X 0,Y 527.913,Z 920.346,A -85,B 0,C 180,E1 24748.264,E2 24748.264} C_VEL
LIN {X 0,Y 527.919,Z 918.001,A -85,B 0,C 180,E1 24746.199,E2 24746.199} C_VEL
LIN {X 0,Y 527.938,Z 914.097,A -85,B 0,C 180,E1 24744.239,E2 24744.239} C_VEL
LIN {X 0,Y 528.01,Z 908.468,A -85,B 0,C 180,E1 24742.273,E2 24742.273} C_VEL
LIN {X 0,Y 528.127,Z 901.427,A -85,B 0,C 180,E1 24740.41,E2 24740.41} C_VEL
LIN {X 0,Y 528.342,Z 892.518,A -85,B 0,C 180,E1 24738.539,E2 24738.539} C_VEL
LIN {X 0,Y 528.655,Z 882.153,A -85,B 0,C 180,E1 24736.771,E2 24736.771} C_VEL
LIN {X 0,Y 529.066,Z 870.352,A -85,B 0,C 180,E1 24735.107,E2 24735.107} C_VEL
LIN {X 0,Y 529.585,Z 857.079,A -85,B 0,C 180,E1 24733.549,E2 24733.549} C_VEL
LIN {X 0,Y 530.195,Z 842.218,A -85,B 0,C 180,E1 24732.098,E2 24732.098} C_VEL
LIN {X 0,Y 530.844,Z 826.235,A -85,B 0,C 180,E1 24730.812,E2 24730.812} C_VEL
LIN {X 0,Y 531.481,Z 809.185,A -85,B 0,C 180,E1 24729.698,E2 24729.698} C_VEL
LIN {X 0,Y 532.082,Z 791.684,A -85,B 0,C 180,E1 24728.788,E2 24728.788} C_VEL
LIN {X 0,Y 532.572,Z 774.032,A -85,B 0,C 180,E1 24728.084,E2 24728.084} C_VEL
LIN {X 0,Y 532.976,Z 755.416,A -85,B 0,C 180,E1 24727.561,E2 24727.561} C_VEL
LIN {X 0,Y 533.222,Z 734.919,A -85,B 0,C 180,E1 24727.203,E2 24727.203} C_VEL
LIN {X 0,Y 534.005,Z 548.204,A -85,B 0,C 180,E1 24724.643,E2 24724.643} C_VEL
LIN {X 0,Y 532.601,Z 538.398,A -85,B 0,C 180,E1 24724.419,E2 24724.419} C_VEL
LIN {X 0,Y 533.804,Z 493.706,A -85,B 0,C 180,E1 24721.102,E2 24721.102} C_VEL
LIN {X 0,Y 534.896,Z 455.777,A -85,B 0,C 180,E1 24718.227,E2 24718.227} C_VEL
LIN {X 0,Y 528.56,Z 437.239,A -85,B 0,C 180,E1 24716.259,E2 24716.259} C_VEL
LIN {X 0,Y 528.523,Z 436.96,A -85,B 0,C 180,E1 24713.152,E2 24713.152} C_VEL
LIN {X 0,Y 528.508,Z 436.962,A -85,B 0,C 180,E1 24709.678,E2 24709.678} C_VEL
LIN {X 0,Y 528.52,Z 436.963,A -85,B 0,C 180,E1 24706.275,E2 24706.275} C_VEL
LIN {X 0,Y 528.519,Z 436.96,A -85,B 0,C 180,E1 24702.776,E2 24702.776} C_VEL
LIN {X 0,Y 528.509,Z 436.959,A -85,B 0,C 180,E1 24699.469,E2 24699.469} C_VEL
LIN {X 0,Y 528.52,Z 436.961,A -85,B 0,C 180,E1 24696.04,E2 24696.04} C_VEL
LIN {X 0,Y 528.519,Z 436.957,A -85,B 0,C 180,E1 24692.498,E2 24692.498} C_VEL
LIN {X 0,Y 528.509,Z 436.957,A -85,B 0,C 180,E1 24689.069,E2 24689.069} C_VEL
LIN {X 0,Y 528.52,Z 436.963,A -85,B 0,C 180,E1 24685.552,E2 24685.552} C_VEL
LIN {X 0,Y 528.517,Z 436.96,A -85,B 0,C 180,E1 24682.115,E2 24682.115} C_VEL
LIN {X 0,Y 528.51,Z 436.956,A -85,B 0,C 180,E1 24678.76,E2 24678.76} C_VEL
LIN {X 0,Y 528.513,Z 436.957,A -85,B 0,C 180,E1 24675.24,E2 24675.24} C_VEL
LIN {X 0,Y 528.516,Z 436.962,A -85,B 0,C 180,E1 24671.789,E2 24671.789} C_VEL
LIN {X 0,Y 528.517,Z 436.956,A -85,B 0,C 180,E1 24668.342,E2 24668.342} C_VEL
LIN {X 0,Y 528.507,Z 436.957,A -85,B 0,C 180,E1 24664.884,E2 24664.884} C_VEL
LIN {X 0,Y 528.517,Z 436.963,A -85,B 0,C 180,E1 24661.517,E2 24661.517} C_VEL
LIN {X 0,Y 528.518,Z 436.957,A -85,B 0,C 180,E1 24658.048,E2 24658.048} C_VEL
LIN {X 0,Y 528.504,Z 436.96,A -85,B 0,C 180,E1 24654.572,E2 24654.572} C_VEL
LIN {X 0,Y 528.521,Z 436.962,A -85,B 0,C 180,E1 24651.185,E2 24651.185} C_VEL
LIN {X 0,Y 528.524,Z 436.958,A -85,B 0,C 180,E1 24647.656,E2 24647.656} C_VEL
LIN {X 0,Y 528.503,Z 436.962,A -85,B 0,C 180,E1 24644.191,E2 24644.191} C_VEL
LIN {X 0,Y 528.521,Z 436.966,A -85,B 0,C 180,E1 24640.736,E2 24640.736} C_VEL
LIN {X 0,Y 528.523,Z 436.96,A -85,B 0,C 180,E1 24637.298,E2 24637.298} C_VEL
LIN {X 0,Y 528.502,Z 436.962,A -85,B 0,C 180,E1 24633.844,E2 24633.844} C_VEL
LIN {X 0,Y 528.518,Z 436.962,A -85,B 0,C 180,E1 24630.411,E2 24630.411} C_VEL
LIN {X 0,Y 528.521,Z 436.962,A -85,B 0,C 180,E1 24626.937,E2 24626.937} C_VEL
LIN {X 0,Y 528.507,Z 436.964,A -85,B 0,C 180,E1 24623.517,E2 24623.517} C_VEL
LIN {X 0,Y 528.5,Z 436.968,A -85,B 0,C 180,E1 24621.685,E2 24621.685} C_VEL
LIN {X 0,Y 527.551,Z 437.332,A -85,B 0,C 180,E1 24621.112,E2 24621.112} C_VEL
LIN {X 0,Y 524.224,Z 439.233,A -85,B 0,C 180,E1 24620.277,E2 24620.277} C_VEL
LIN {X 0,Y 522.339,Z 441.652,A -85,B 0,C 180,E1 24619.696,E2 24619.696} C_VEL
LIN {X 0,Y 522.269,Z 444.053,A -85,B 0,C 180,E1 24619.278,E2 24619.278} C_VEL
LIN {X 0,Y 524.997,Z 454.491,A -85,B 0,C 180,E1 24617.756,E2 24617.756} C_VEL
LIN {X 0,Y 523.796,Z 483.631,A -85,B 0,C 180,E1 24614.166,E2 24614.166} C_VEL
LIN {X 0,Y 522.877,Z 511.673,A -85,B 0,C 180,E1 24610.778,E2 24610.778} C_VEL
LIN {X 0,Y 521.899,Z 541.876,A -85,B 0,C 180,E1 24607.157,E2 24607.157} C_VEL
LIN {X 0,Y 521.604,Z 556.7,A -85,B 0,C 180,E1 24605.461,E2 24605.461} C_VEL
LIN {X 0,Y 523.027,Z 567.67,A -85,B 0,C 180,E1 24605.231,E2 24605.231} C_VEL
LIN {X 0,Y 522.355,Z 669.735,A -85,B 0,C 180,E1 24603.754,E2 24603.754} C_VEL
LIN {X 0,Y 522.169,Z 684.576,A -85,B 0,C 180,E1 24603.336,E2 24603.336} C_VEL
LIN {X 0,Y 521.862,Z 699.068,A -85,B 0,C 180,E1 24602.704,E2 24602.704} C_VEL
LIN {X 0,Y 521.507,Z 711.721,A -85,B 0,C 180,E1 24601.949,E2 24601.949} C_VEL
LIN {X 0,Y 521.105,Z 724.583,A -85,B 0,C 180,E1 24600.943,E2 24600.943} C_VEL
LIN {X 0,Y 520.769,Z 735.899,A -85,B 0,C 180,E1 24599.792,E2 24599.792} C_VEL
LIN {X 0,Y 520.482,Z 745.346,A -85,B 0,C 180,E1 24598.577,E2 24598.577} C_VEL
LIN {X 0,Y 520.255,Z 754.025,A -85,B 0,C 180,E1 24597.148,E2 24597.148} C_VEL
LIN {X 0,Y 520.085,Z 760.989,A -85,B 0,C 180,E1 24595.623,E2 24595.623} C_VEL
LIN {X 0,Y 519.993,Z 766.151,A -85,B 0,C 180,E1 24594.057,E2 24594.057} C_VEL
LIN {X 0,Y 519.952,Z 769.725,A -85,B 0,C 180,E1 24592.38,E2 24592.38} C_VEL
LIN {X 0,Y 519.941,Z 771.463,A -85,B 0,C 180,E1 24590.604,E2 24590.604} C_VEL
LIN {X 0,Y 519.94,Z 771.189,A -85,B 0,C 180,E1 24588.848,E2 24588.848} C_VEL
LIN {X 0,Y 519.954,Z 769.184,A -85,B 0,C 180,E1 24587.226,E2 24587.226} C_VEL
LIN {X 0,Y 520.002,Z 765.319,A -85,B 0,C 180,E1 24585.565,E2 24585.565} C_VEL
LIN {X 0,Y 520.114,Z 759.277,A -85,B 0,C 180,E1 24583.878,E2 24583.878} C_VEL
LIN {X 0,Y 520.302,Z 751.461,A -85,B 0,C 180,E1 24582.316,E2 24582.316} C_VEL
LIN {X 0,Y 520.542,Z 742.554,A -85,B 0,C 180,E1 24580.962,E2 24580.962} C_VEL
LIN {X 0,Y 520.859,Z 732.179,A -85,B 0,C 180,E1 24579.725,E2 24579.725} C_VEL
LIN {X 0,Y 521.217,Z 720.119,A -85,B 0,C 180,E1 24578.605,E2 24578.605} C_VEL
LIN {X 0,Y 521.606,Z 707.037,A -85,B 0,C 180,E1 24577.677,E2 24577.677} C_VEL
LIN {X 0,Y 521.926,Z 694.219,A -85,B 0,C 180,E1 24576.987,E2 24576.987} C_VEL
LIN {X 0,Y 522.22,Z 678.898,A -85,B 0,C 180,E1 24576.407,E2 24576.407} C_VEL
LIN {X 0,Y 522.391,Z 663.038,A -85,B 0,C 180,E1 24576.053,E2 24576.053} C_VEL
LIN {X 0,Y 522.738,Z 564.074,A -85,B 0,C 180,E1 24574.647,E2 24574.647} C_VEL
LIN {X 0,Y 521.545,Z 556.22,A -85,B 0,C 180,E1 24574.453,E2 24574.453} C_VEL
LIN {X 0,Y 522.167,Z 529.462,A -85,B 0,C 180,E1 24571.316,E2 24571.316} C_VEL
LIN {X 0,Y 523.113,Z 500.203,A -85,B 0,C 180,E1 24567.809,E2 24567.809} C_VEL
LIN {X 0,Y 524.096,Z 472.201,A -85,B 0,C 180,E1 24564.416,E2 24564.416} C_VEL
LIN {X 0,Y 524.732,Z 453.606,A -85,B 0,C 180,E1 24562.114,E2 24562.114} C_VEL
LIN {X 0,Y 520.589,Z 438.056,A -85,B 0,C 180,E1 24559.822,E2 24559.822} C_VEL
LIN {X 0,Y 520.516,Z 437.957,A -85,B 0,C 180,E1 24556.446,E2 24556.446} C_VEL
LIN {X 0,Y 520.528,Z 437.957,A -85,B 0,C 180,E1 24553.024,E2 24553.024} C_VEL
LIN {X 0,Y 520.553,Z 437.954,A -85,B 0,C 180,E1 24549.773,E2 24549.773} C_VEL
LIN {X 0,Y 520.505,Z 437.941,A -85,B 0,C 180,E1 24546.449,E2 24546.449} C_VEL
LIN {X 0,Y 520.554,Z 437.955,A -85,B 0,C 180,E1 24543.168,E2 24543.168} C_VEL
LIN {X 0,Y 520.511,Z 437.957,A -85,B 0,C 180,E1 24540.036,E2 24540.036} C_VEL
LIN {X 0,Y 520.506,Z 437.956,A -85,B 0,C 180,E1 24536.48,E2 24536.48} C_VEL
LIN {X 0,Y 520.57,Z 437.949,A -85,B 0,C 180,E1 24533.183,E2 24533.183} C_VEL
LIN {X 0,Y 520.514,Z 437.957,A -85,B 0,C 180,E1 24529.865,E2 24529.865} C_VEL
LIN {X 0,Y 520.518,Z 437.953,A -85,B 0,C 180,E1 24526.401,E2 24526.401} C_VEL
LIN {X 0,Y 520.573,Z 437.951,A -85,B 0,C 180,E1 24523.125,E2 24523.125} C_VEL
LIN {X 0,Y 520.515,Z 437.951,A -85,B 0,C 180,E1 24519.91,E2 24519.91} C_VEL
LIN {X 0,Y 520.551,Z 437.95,A -85,B 0,C 180,E1 24516.544,E2 24516.544} C_VEL
LIN {X 0,Y 520.541,Z 437.944,A -85,B 0,C 180,E1 24513.323,E2 24513.323} C_VEL
LIN {X 0,Y 520.525,Z 437.954,A -85,B 0,C 180,E1 24509.962,E2 24509.962} C_VEL
LIN {X 0,Y 520.584,Z 437.939,A -85,B 0,C 180,E1 24506.708,E2 24506.708} C_VEL
LIN {X 0,Y 520.535,Z 437.952,A -85,B 0,C 180,E1 24503.341,E2 24503.341} C_VEL
LIN {X 0,Y 520.535,Z 437.948,A -85,B 0,C 180,E1 24499.876,E2 24499.876} C_VEL
LIN {X 0,Y 520.587,Z 437.943,A -85,B 0,C 180,E1 24496.515,E2 24496.515} C_VEL
LIN {X 0,Y 520.539,Z 437.954,A -85,B 0,C 180,E1 24493.214,E2 24493.214} C_VEL
LIN {X 0,Y 520.543,Z 437.941,A -85,B 0,C 180,E1 24489.732,E2 24489.732} C_VEL
LIN {X 0,Y 520.59,Z 437.95,A -85,B 0,C 180,E1 24486.396,E2 24486.396} C_VEL
LIN {X 0,Y 520.547,Z 437.953,A -85,B 0,C 180,E1 24482.973,E2 24482.973} C_VEL
LIN {X 0,Y 520.544,Z 437.94,A -85,B 0,C 180,E1 24479.45,E2 24479.45} C_VEL
LIN {X 0,Y 520.586,Z 437.95,A -85,B 0,C 180,E1 24476.035,E2 24476.035} C_VEL
LIN {X 0,Y 520.564,Z 437.946,A -85,B 0,C 180,E1 24472.606,E2 24472.606} C_VEL
LIN {X 0,Y 520.547,Z 437.95,A -85,B 0,C 180,E1 24469.15,E2 24469.15} C_VEL
LIN {X 0,Y 520.587,Z 437.94,A -85,B 0,C 180,E1 24465.769,E2 24465.769} C_VEL
LIN {X 0,Y 520.579,Z 437.953,A -85,B 0,C 180,E1 24462.299,E2 24462.299} C_VEL
LIN {X 0,Y 520.553,Z 437.946,A -85,B 0,C 180,E1 24458.832,E2 24458.832} C_VEL
LIN {X 0,Y 520.579,Z 437.948,A -85,B 0,C 180,E1 24455.368,E2 24455.368} C_VEL
LIN {X 0,Y 520.587,Z 437.951,A -85,B 0,C 180,E1 24451.93,E2 24451.93} C_VEL
LIN {X 0,Y 520.561,Z 437.95,A -85,B 0,C 180,E1 24448.504,E2 24448.504} C_VEL
LIN {X 0,Y 520.57,Z 437.947,A -85,B 0,C 180,E1 24444.95,E2 24444.95} C_VEL
LIN {X 0,Y 520.581,Z 437.948,A -85,B 0,C 180,E1 24441.516,E2 24441.516} C_VEL
LIN {X 0,Y 520.579,Z 437.953,A -85,B 0,C 180,E1 24438.013,E2 24438.013} C_VEL
LIN {X 0,Y 520.566,Z 437.948,A -85,B 0,C 180,E1 24434.512,E2 24434.512} C_VEL
LIN {X 0,Y 520.589,Z 437.949,A -85,B 0,C 180,E1 24430.992,E2 24430.992} C_VEL
LIN {X 0,Y 520.581,Z 437.953,A -85,B 0,C 180,E1 24427.507,E2 24427.507} C_VEL
LIN {X 0,Y 520.605,Z 438.194,A -85,B 0,C 180,E1 24424.203,E2 24424.203} C_VEL
LIN {X 0,Y 524.715,Z 450.061,A -85,B 0,C 180,E1 24422.894,E2 24422.894} C_VEL
LIN {X 0,Y 527.619,Z 458.801,A -85,B 0,C 180,E1 24421.983,E2 24421.983} C_VEL
LIN {X 0,Y 526.441,Z 493.052,A -85,B 0,C 180,E1 24419.335,E2 24419.335} C_VEL
LIN {X 0,Y 525.039,Z 538.986,A -85,B 0,C 180,E1 24415.87,E2 24415.87} C_VEL
LIN {X 0,Y 526.696,Z 552.013,A -85,B 0,C 180,E1 24415.606,E2 24415.606} C_VEL
LIN {X 0,Y 525.491,Z 747.611,A -85,B 0,C 180,E1 24412.866,E2 24412.866} C_VEL
LIN {X 0,Y 525.082,Z 766.877,A -85,B 0,C 180,E1 24412.392,E2 24412.392} C_VEL
LIN {X 0,Y 524.569,Z 785.409,A -85,B 0,C 180,E1 24411.731,E2 24411.731} C_VEL
LIN {X 0,Y 524.019,Z 802.932,A -85,B 0,C 180,E1 24410.904,E2 24410.904} C_VEL
LIN {X 0,Y 523.375,Z 820.152,A -85,B 0,C 180,E1 24409.88,E2 24409.88} C_VEL
LIN {X 0,Y 522.808,Z 834.98,A -85,B 0,C 180,E1 24408.795,E2 24408.795} C_VEL
LIN {X 0,Y 522.123,Z 849.994,A -85,B 0,C 180,E1 24407.44,E2 24407.44} C_VEL
LIN {X 0,Y 521.494,Z 864.017,A -85,B 0,C 180,E1 24405.913,E2 24405.913} C_VEL
LIN {X 0,Y 520.962,Z 876.702,A -85,B 0,C 180,E1 24404.252,E2 24404.252} C_VEL
LIN {X 0,Y 520.562,Z 887.591,A -85,B 0,C 180,E1 24402.536,E2 24402.536} C_VEL
LIN {X 0,Y 520.261,Z 897.477,A -85,B 0,C 180,E1 24400.632,E2 24400.632} C_VEL
LIN {X 0,Y 520.067,Z 905.77,A -85,B 0,C 180,E1 24398.625,E2 24398.625} C_VEL
LIN {X 0,Y 519.967,Z 912.108,A -85,B 0,C 180,E1 24396.626,E2 24396.626} C_VEL
LIN {X 0,Y 519.926,Z 916.876,A -85,B 0,C 180,E1 24394.522,E2 24394.522} C_VEL
LIN {X 0,Y 519.912,Z 919.793,A -85,B 0,C 180,E1 24392.425,E2 24392.425} C_VEL
LIN {X 0,Y 519.908,Z 920.939,A -85,B 0,C 180,E1 24390.331,E2 24390.331} C_VEL
LIN {X 0,Y 519.913,Z 920.346,A -85,B 0,C 180,E1 24388.237,E2 24388.237} C_VEL
LIN {X 0,Y 519.917,Z 918.16,A -85,B 0,C 180,E1 24386.251,E2 24386.251} C_VEL
LIN {X 0,Y 519.94,Z 914.351,A -85,B 0,C 180,E1 24384.261,E2 24384.261} C_VEL
LIN {X 0,Y 520.018,Z 908.822,A -85,B 0,C 180,E1 24382.265,E2 24382.265} C_VEL
LIN {X 0,Y 520.159,Z 901.427,A -85,B 0,C 180,E1 24380.261,E2 24380.261} C_VEL
LIN {X 0,Y 520.402,Z 892.517,A -85,B 0,C 180,E1 24378.362,E2 24378.362} C_VEL
LIN {X 0,Y 520.756,Z 882.152,A -85,B 0,C 180,E1 24376.566,E2 24376.566} C_VEL
LIN {X 0,Y 521.224,Z 870.351,A -85,B 0,C 180,E1 24374.877,E2 24374.877} C_VEL
LIN {X 0,Y 521.802,Z 857.078,A -85,B 0,C 180,E1 24373.296,E2 24373.296} C_VEL
LIN {X 0,Y 522.483,Z 842.217,A -85,B 0,C 180,E1 24371.825,E2 24371.825} C_VEL
LIN {X 0,Y 523.115,Z 827.562,A -85,B 0,C 180,E1 24370.633,E2 24370.633} C_VEL
LIN {X 0,Y 523.713,Z 811.043,A -85,B 0,C 180,E1 24369.551,E2 24369.551} C_VEL
LIN {X 0,Y 524.312,Z 793.757,A -85,B 0,C 180,E1 24368.64,E2 24368.64} C_VEL
LIN {X 0,Y 524.84,Z 775.672,A -85,B 0,C 180,E1 24367.898,E2 24367.898} C_VEL
LIN {X 0,Y 525.308,Z 756.489,A -85,B 0,C 180,E1 24367.33,E2 24367.33} C_VEL
LIN {X 0,Y 525.593,Z 736.43,A -85,B 0,C 180,E1 24366.958,E2 24366.958} C_VEL
LIN {X 0,Y 526.486,Z 549.202,A -85,B 0,C 180,E1 24364.358,E2 24364.358} C_VEL
LIN {X 0,Y 525.007,Z 538.538,A -85,B 0,C 180,E1 24364.113,E2 24364.113} C_VEL
LIN {X 0,Y 526.448,Z 492.47,A -85,B 0,C 180,E1 24360.624,E2 24360.624} C_VEL
LIN {X 0,Y 527.6,Z 458.638,A -85,B 0,C 180,E1 24358.01,E2 24358.01} C_VEL
LIN {X 0,Y 520.636,Z 438.372,A -85,B 0,C 180,E1 24355.824,E2 24355.824} C_VEL
LIN {X 0,Y 520.582,Z 437.955,A -85,B 0,C 180,E1 24355.22,E2 24355.22} C_VEL
LIN {X 0,Y 520.571,Z 437.951,A -85,B 0,C 180,E1 24351.773,E2 24351.773} C_VEL
LIN {X 0,Y 520.578,Z 437.954,A -85,B 0,C 180,E1 24348.343,E2 24348.343} C_VEL
LIN {X 0,Y 520.581,Z 437.946,A -85,B 0,C 180,E1 24344.82,E2 24344.82} C_VEL
LIN {X 0,Y 520.571,Z 437.951,A -85,B 0,C 180,E1 24341.324,E2 24341.324} C_VEL
LIN {X 0,Y 520.583,Z 437.955,A -85,B 0,C 180,E1 24337.784,E2 24337.784} C_VEL
LIN {X 0,Y 520.577,Z 437.951,A -85,B 0,C 180,E1 24334.247,E2 24334.247} C_VEL
LIN {X 0,Y 520.586,Z 437.946,A -85,B 0,C 180,E1 24330.723,E2 24330.723} C_VEL
LIN {X 0,Y 520.569,Z 437.951,A -85,B 0,C 180,E1 24327.202,E2 24327.202} C_VEL
LIN {X 0,Y 520.583,Z 437.946,A -85,B 0,C 180,E1 24323.787,E2 24323.787} C_VEL
LIN {X 0,Y 520.581,Z 437.946,A -85,B 0,C 180,E1 24320.225,E2 24320.225} C_VEL
LIN {X 0,Y 520.57,Z 437.949,A -85,B 0,C 180,E1 24316.744,E2 24316.744} C_VEL
LIN {X 0,Y 520.577,Z 437.953,A -85,B 0,C 180,E1 24313.212,E2 24313.212} C_VEL
LIN {X 0,Y 520.577,Z 437.946,A -85,B 0,C 180,E1 24309.731,E2 24309.731} C_VEL
LIN {X 0,Y 520.579,Z 437.947,A -85,B 0,C 180,E1 24306.285,E2 24306.285} C_VEL
LIN {X 0,Y 520.566,Z 437.952,A -85,B 0,C 180,E1 24302.752,E2 24302.752} C_VEL
LIN {X 0,Y 520.582,Z 437.944,A -85,B 0,C 180,E1 24299.339,E2 24299.339} C_VEL
LIN {X 0,Y 520.582,Z 437.945,A -85,B 0,C 180,E1 24295.814,E2 24295.814} C_VEL
LIN {X 0,Y 520.564,Z 437.95,A -85,B 0,C 180,E1 24292.346,E2 24292.346} C_VEL
LIN {X 0,Y 520.582,Z 437.952,A -85,B 0,C 180,E1 24288.926,E2 24288.926} C_VEL
LIN {X 0,Y 520.581,Z 437.944,A -85,B 0,C 180,E1 24285.427,E2 24285.427} C_VEL
LIN {X 0,Y 520.567,Z 437.946,A -85,B 0,C 180,E1 24281.987,E2 24281.987} C_VEL
LIN {X 0,Y 520.574,Z 437.951,A -85,B 0,C 180,E1 24278.478,E2 24278.478} C_VEL
LIN {X 0,Y 520.581,Z 437.947,A -85,B 0,C 180,E1 24275.004,E2 24275.004} C_VEL
LIN {X 0,Y 520.578,Z 437.949,A -85,B 0,C 180,E1 24271.554,E2 24271.554} C_VEL
LIN {X 0,Y 520.566,Z 437.951,A -85,B 0,C 180,E1 24268.098,E2 24268.098} C_VEL
LIN {X 0,Y 520.583,Z 437.954,A -85,B 0,C 180,E1 24264.681,E2 24264.681} C_VEL
LIN {X 0,Y 520.584,Z 437.954,A -85,B 0,C 180,E1 24261.234,E2 24261.234} C_VEL
LIN {X 0,Y 520.62,Z 438.259,A -85,B 0,C 180,E1 24260.162,E2 24260.162} C_VEL
LIN {X 0,Y 522.269,Z 444.053,A -85,B 0,C 180,E1 24259.278,E2 24259.278} C_VEL
LIN {X 0,Y 522.605,Z 448.249,A -85,B 0,C 180,E1 24258.715,E2 24258.715} C_VEL
LIN {X 0,Y 521.156,Z 454.412,A -85,B 0,C 180,E1 24258.02,E2 24258.02} C_VEL
LIN {X 0,Y 517.422,Z 465.598,A -85,B 0,C 180,E1 24256.828,E2 24256.828} C_VEL
LIN {X 0,Y 516.978,Z 468.685,A -85,B 0,C 180,E1 24256.46,E2 24256.46} C_VEL
LIN {X 0,Y 515.828,Z 497.073,A -85,B 0,C 180,E1 24252.94,E2 24252.94} C_VEL
LIN {X 0,Y 514.744,Z 526.375,A -85,B 0,C 180,E1 24249.367,E2 24249.367} C_VEL
LIN {X 0,Y 513.866,Z 556.121,A -85,B 0,C 180,E1 24245.819,E2 24245.819} C_VEL
LIN {X 0,Y 515.549,Z 567.84,A -85,B 0,C 180,E1 24245.544,E2 24245.544} C_VEL
LIN {X 0,Y 514.78,Z 670.592,A -85,B 0,C 180,E1 24244.027,E2 24244.027} C_VEL
LIN {X 0,Y 514.58,Z 685.333,A -85,B 0,C 180,E1 24243.603,E2 24243.603} C_VEL
LIN {X 0,Y 514.257,Z 699.395,A -85,B 0,C 180,E1 24242.983,E2 24242.983} C_VEL
LIN {X 0,Y 513.871,Z 712.201,A -85,B 0,C 180,E1 24242.217,E2 24242.217} C_VEL
LIN {X 0,Y 513.422,Z 725.132,A -85,B 0,C 180,E1 24241.199,E2 24241.199} C_VEL
LIN {X 0,Y 513.044,Z 736.327,A -85,B 0,C 180,E1 24240.057,E2 24240.057} C_VEL
LIN {X 0,Y 512.708,Z 746.107,A -85,B 0,C 180,E1 24238.795,E2 24238.795} C_VEL
LIN {X 0,Y 512.428,Z 755.135,A -85,B 0,C 180,E1 24237.293,E2 24237.293} C_VEL
LIN {X 0,Y 512.217,Z 762.355,A -85,B 0,C 180,E1 24235.68,E2 24235.68} C_VEL
LIN {X 0,Y 512.102,Z 767.458,A -85,B 0,C 180,E1 24234.083,E2 24234.083} C_VEL
LIN {X 0,Y 512.05,Z 770.789,A -85,B 0,C 180,E1 24232.502,E2 24232.502} C_VEL
LIN {X 0,Y 512.028,Z 772.589,A -85,B 0,C 180,E1 24230.698,E2 24230.698} C_VEL
LIN {X 0,Y 512.025,Z 772.473,A -85,B 0,C 180,E1 24229.033,E2 24229.033} C_VEL
LIN {X 0,Y 512.045,Z 770.705,A -85,B 0,C 180,E1 24227.383,E2 24227.383} C_VEL
LIN {X 0,Y 512.102,Z 766.867,A -85,B 0,C 180,E1 24225.631,E2 24225.631} C_VEL
LIN {X 0,Y 512.221,Z 761.363,A -85,B 0,C 180,E1 24224.007,E2 24224.007} C_VEL
LIN {X 0,Y 512.417,Z 754.393,A -85,B 0,C 180,E1 24222.509,E2 24222.509} C_VEL
LIN {X 0,Y 512.7,Z 745.246,A -85,B 0,C 180,E1 24221.018,E2 24221.018} C_VEL
LIN {X 0,Y 513.073,Z 734.254,A -85,B 0,C 180,E1 24219.648,E2 24219.648} C_VEL
LIN {X 0,Y 513.461,Z 722.469,A -85,B 0,C 180,E1 24218.511,E2 24218.511} C_VEL
LIN {X 0,Y 513.867,Z 710.433,A -85,B 0,C 180,E1 24217.603,E2 24217.603} C_VEL
LIN {X 0,Y 514.256,Z 696.568,A -85,B 0,C 180,E1 24216.811,E2 24216.811} C_VEL
LIN {X 0,Y 514.56,Z 682.104,A -85,B 0,C 180,E1 24216.226,E2 24216.226} C_VEL
LIN {X 0,Y 514.767,Z 667.289,A -85,B 0,C 180,E1 24215.844,E2 24215.844} C_VEL
LIN {X 0,Y 515.199,Z 564.796,A -85,B 0,C 180,E1 24214.351,E2 24214.351} C_VEL
LIN {X 0,Y 513.803,Z 556.022,A -85,B 0,C 180,E1 24214.129,E2 24214.129} C_VEL
LIN {X 0,Y 514.564,Z 527.857,A -85,B 0,C 180,E1 24210.779,E2 24210.779} C_VEL
LIN {X 0,Y 515.559,Z 499.486,A -85,B 0,C 180,E1 24207.332,E2 24207.332} C_VEL
LIN {X 0,Y 516.711,Z 470.605,A -85,B 0,C 180,E1 24203.779,E2 24203.779} C_VEL
LIN {X 0,Y 517.303,Z 456.401,A -85,B 0,C 180,E1 24202,E2 24202} C_VEL
LIN {X 0,Y 512.639,Z 439.069,A -85,B 0,C 180,E1 24199.425,E2 24199.425} C_VEL
LIN {X 0,Y 512.596,Z 438.946,A -85,B 0,C 180,E1 24196.118,E2 24196.118} C_VEL
LIN {X 0,Y 512.575,Z 438.946,A -85,B 0,C 180,E1 24192.752,E2 24192.752} C_VEL
LIN {X 0,Y 512.636,Z 438.946,A -85,B 0,C 180,E1 24189.425,E2 24189.425} C_VEL
LIN {X 0,Y 512.571,Z 438.928,A -85,B 0,C 180,E1 24186.184,E2 24186.184} C_VEL
LIN {X 0,Y 512.575,Z 438.944,A -85,B 0,C 180,E1 24182.716,E2 24182.716} C_VEL
LIN {X 0,Y 512.614,Z 438.946,A -85,B 0,C 180,E1 24179.527,E2 24179.527} C_VEL
LIN {X 0,Y 512.564,Z 438.945,A -85,B 0,C 180,E1 24176.202,E2 24176.202} C_VEL
LIN {X 0,Y 512.596,Z 438.941,A -85,B 0,C 180,E1 24172.794,E2 24172.794} C_VEL
LIN {X 0,Y 512.603,Z 438.946,A -85,B 0,C 180,E1 24169.493,E2 24169.493} C_VEL
LIN {X 0,Y 512.572,Z 438.942,A -85,B 0,C 180,E1 24166.172,E2 24166.172} C_VEL
LIN {X 0,Y 512.625,Z 438.936,A -85,B 0,C 180,E1 24162.829,E2 24162.829} C_VEL
LIN {X 0,Y 512.587,Z 438.94,A -85,B 0,C 180,E1 24159.602,E2 24159.602} C_VEL
LIN {X 0,Y 512.582,Z 438.939,A -85,B 0,C 180,E1 24156.093,E2 24156.093} C_VEL
LIN {X 0,Y 512.639,Z 438.939,A -85,B 0,C 180,E1 24152.702,E2 24152.702} C_VEL
LIN {X 0,Y 512.593,Z 438.944,A -85,B 0,C 180,E1 24149.443,E2 24149.443} C_VEL
LIN {X 0,Y 512.588,Z 438.928,A -85,B 0,C 180,E1 24145.909,E2 24145.909} C_VEL
LIN {X 0,Y 512.652,Z 438.941,A -85,B 0,C 180,E1 24142.596,E2 24142.596} C_VEL
LIN {X 0,Y 512.599,Z 438.939,A -85,B 0,C 180,E1 24139.248,E2 24139.248} C_VEL
LIN {X 0,Y 512.595,Z 438.935,A -85,B 0,C 180,E1 24135.732,E2 24135.732} C_VEL
LIN {X 0,Y 512.647,Z 438.938,A -85,B 0,C 180,E1 24132.389,E2 24132.389} C_VEL
LIN {X 0,Y 512.61,Z 438.931,A -85,B 0,C 180,E1 24128.977,E2 24128.977} C_VEL
LIN {X 0,Y 512.602,Z 438.939,A -85,B 0,C 180,E1 24125.485,E2 24125.485} C_VEL
LIN {X 0,Y 512.64,Z 438.93,A -85,B 0,C 180,E1 24122.012,E2 24122.012} C_VEL
LIN {X 0,Y 512.637,Z 438.933,A -85,B 0,C 180,E1 24118.547,E2 24118.547} C_VEL
LIN {X 0,Y 512.606,Z 438.941,A -85,B 0,C 180,E1 24115.077,E2 24115.077} C_VEL
LIN {X 0,Y 512.626,Z 438.928,A -85,B 0,C 180,E1 24111.589,E2 24111.589} C_VEL
LIN {X 0,Y 512.647,Z 438.942,A -85,B 0,C 180,E1 24108.183,E2 24108.183} C_VEL
LIN {X 0,Y 512.614,Z 438.933,A -85,B 0,C 180,E1 24104.733,E2 24104.733} C_VEL
LIN {X 0,Y 512.623,Z 438.938,A -85,B 0,C 180,E1 24101.227,E2 24101.227} C_VEL
LIN {X 0,Y 512.647,Z 438.936,A -85,B 0,C 180,E1 24097.767,E2 24097.767} C_VEL
LIN {X 0,Y 512.634,Z 438.943,A -85,B 0,C 180,E1 24094.304,E2 24094.304} C_VEL
LIN {X 0,Y 512.62,Z 438.939,A -85,B 0,C 180,E1 24090.816,E2 24090.816} C_VEL
LIN {X 0,Y 512.646,Z 438.936,A -85,B 0,C 180,E1 24087.413,E2 24087.413} C_VEL
LIN {X 0,Y 512.645,Z 438.938,A -85,B 0,C 180,E1 24083.849,E2 24083.849} C_VEL
LIN {X 0,Y 512.625,Z 438.938,A -85,B 0,C 180,E1 24080.372,E2 24080.372} C_VEL
LIN {X 0,Y 512.637,Z 438.937,A -85,B 0,C 180,E1 24076.841,E2 24076.841} C_VEL
LIN {X 0,Y 512.641,Z 438.941,A -85,B 0,C 180,E1 24073.323,E2 24073.323} C_VEL
LIN {X 0,Y 512.649,Z 438.939,A -85,B 0,C 180,E1 24069.772,E2 24069.772} C_VEL
LIN {X 0,Y 512.631,Z 438.94,A -85,B 0,C 180,E1 24066.227,E2 24066.227} C_VEL
LIN {X 0,Y 512.683,Z 439.226,A -85,B 0,C 180,E1 24064.658,E2 24064.658} C_VEL
LIN {X 0,Y 520.303,Z 461.373,A -85,B 0,C 180,E1 24062.233,E2 24062.233} C_VEL
LIN {X 0,Y 519.023,Z 494.659,A -85,B 0,C 180,E1 24059.613,E2 24059.613} C_VEL
LIN {X 0,Y 517.478,Z 539.254,A -85,B 0,C 180,E1 24056.185,E2 24056.185} C_VEL
LIN {X 0,Y 519.203,Z 553.009,A -85,B 0,C 180,E1 24055.903,E2 24055.903} C_VEL
LIN {X 0,Y 517.883,Z 747.15,A -85,B 0,C 180,E1 24053.146,E2 24053.146} C_VEL
LIN {X 0,Y 517.437,Z 766.215,A -85,B 0,C 180,E1 24052.671,E2 24052.671} C_VEL
LIN {X 0,Y 516.876,Z 784.719,A -85,B 0,C 180,E1 24052.002,E2 24052.002} C_VEL
LIN {X 0,Y 516.291,Z 802.052,A -85,B 0,C 180,E1 24051.173,E2 24051.173} C_VEL
LIN {X 0,Y 515.586,Z 819.273,A -85,B 0,C 180,E1 24050.134,E2 24050.134} C_VEL
LIN {X 0,Y 514.915,Z 835.603,A -85,B 0,C 180,E1 24048.922,E2 24048.922} C_VEL
LIN {X 0,Y 514.228,Z 850.988,A -85,B 0,C 180,E1 24047.541,E2 24047.541} C_VEL
LIN {X 0,Y 513.628,Z 864.84,A -85,B 0,C 180,E1 24046.047,E2 24046.047} C_VEL
LIN {X 0,Y 513.124,Z 876.138,A -85,B 0,C 180,E1 24044.559,E2 24044.559} C_VEL
LIN {X 0,Y 512.666,Z 887.222,A -85,B 0,C 180,E1 24042.798,E2 24042.798} C_VEL
LIN {X 0,Y 512.325,Z 896.962,A -85,B 0,C 180,E1 24040.913,E2 24040.913} C_VEL
LIN {X 0,Y 512.104,Z 904.96,A -85,B 0,C 180,E1 24038.986,E2 24038.986} C_VEL
LIN {X 0,Y 511.986,Z 911.502,A -85,B 0,C 180,E1 24036.955,E2 24036.955} C_VEL
LIN {X 0,Y 511.927,Z 916.256,A -85,B 0,C 180,E1 24034.93,E2 24034.93} C_VEL
LIN {X 0,Y 511.911,Z 919.338,A -85,B 0,C 180,E1 24032.911,E2 24032.911} C_VEL
LIN {X 0,Y 511.91,Z 920.826,A -85,B 0,C 180,E1 24030.896,E2 24030.896} C_VEL
LIN {X 0,Y 511.906,Z 920.752,A -85,B 0,C 180,E1 24028.881,E2 24028.881} C_VEL
LIN {X 0,Y 511.913,Z 918.956,A -85,B 0,C 180,E1 24026.753,E2 24026.753} C_VEL
LIN {X 0,Y 511.936,Z 915.367,A -85,B 0,C 180,E1 24024.621,E2 24024.621} C_VEL
LIN {X 0,Y 512.003,Z 910.234,A -85,B 0,C 180,E1 24022.595,E2 24022.595} C_VEL
LIN {X 0,Y 512.15,Z 903.26,A -85,B 0,C 180,E1 24020.562,E2 24020.562} C_VEL
LIN {X 0,Y 512.393,Z 894.81,A -85,B 0,C 180,E1 24018.634,E2 24018.634} C_VEL
LIN {X 0,Y 512.754,Z 884.953,A -85,B 0,C 180,E1 24016.812,E2 24016.812} C_VEL
LIN {X 0,Y 513.231,Z 873.599,A -85,B 0,C 180,E1 24015.081,E2 24015.081} C_VEL
LIN {X 0,Y 513.759,Z 861.942,A -85,B 0,C 180,E1 24013.609,E2 24013.609} C_VEL
LIN {X 0,Y 514.381,Z 847.423,A -85,B 0,C 180,E1 24012.114,E2 24012.114} C_VEL
LIN {X 0,Y 515.064,Z 831.973,A -85,B 0,C 180,E1 24010.79,E2 24010.79} C_VEL
LIN {X 0,Y 515.715,Z 815.67,A -85,B 0,C 180,E1 24009.634,E2 24009.634} C_VEL
LIN {X 0,Y 516.41,Z 798.287,A -85,B 0,C 180,E1 24008.638,E2 24008.638} C_VEL
LIN {X 0,Y 517.012,Z 779.953,A -85,B 0,C 180,E1 24007.815,E2 24007.815} C_VEL
LIN {X 0,Y 517.53,Z 761.189,A -85,B 0,C 180,E1 24007.195,E2 24007.195} C_VEL
LIN {X 0,Y 517.915,Z 741.712,A -85,B 0,C 180,E1 24006.77,E2 24006.77} C_VEL
LIN {X 0,Y 518.976,Z 550.186,A -85,B 0,C 180,E1 24004.065,E2 24004.065} C_VEL
LIN {X 0,Y 517.435,Z 539.209,A -85,B 0,C 180,E1 24003.829,E2 24003.829} C_VEL
LIN {X 0,Y 519.004,Z 492.799,A -85,B 0,C 180,E1 24000.272,E2 24000.272} C_VEL
LIN {X 0,Y 520.188,Z 461.095,A -85,B 0,C 180,E1 23997.75,E2 23997.75} C_VEL
LIN {X 0,Y 513.419,Z 441.56,A -85,B 0,C 180,E1 23995.614,E2 23995.614} C_VEL
LIN {X 0,Y 512.67,Z 439.132,A -85,B 0,C 180,E1 23995.286,E2 23995.286} C_VEL
LIN {X 0,Y 512.634,Z 438.94,A -85,B 0,C 180,E1 23991.809,E2 23991.809} C_VEL
LIN {X 0,Y 512.64,Z 438.943,A -85,B 0,C 180,E1 23988.311,E2 23988.311} C_VEL
LIN {X 0,Y 512.641,Z 438.936,A -85,B 0,C 180,E1 23984.757,E2 23984.757} C_VEL
LIN {X 0,Y 512.635,Z 438.939,A -85,B 0,C 180,E1 23981.242,E2 23981.242} C_VEL
LIN {X 0,Y 512.637,Z 438.943,A -85,B 0,C 180,E1 23977.639,E2 23977.639} C_VEL
LIN {X 0,Y 512.64,Z 438.94,A -85,B 0,C 180,E1 23974.175,E2 23974.175} C_VEL
LIN {X 0,Y 512.647,Z 438.936,A -85,B 0,C 180,E1 23970.6,E2 23970.6} C_VEL
LIN {X 0,Y 512.631,Z 438.939,A -85,B 0,C 180,E1 23967.155,E2 23967.155} C_VEL
LIN {X 0,Y 512.646,Z 438.934,A -85,B 0,C 180,E1 23963.689,E2 23963.689} C_VEL
LIN {X 0,Y 512.642,Z 438.936,A -85,B 0,C 180,E1 23960.195,E2 23960.195} C_VEL
LIN {X 0,Y 512.632,Z 438.938,A -85,B 0,C 180,E1 23956.732,E2 23956.732} C_VEL
LIN {X 0,Y 512.637,Z 438.942,A -85,B 0,C 180,E1 23953.191,E2 23953.191} C_VEL
LIN {X 0,Y 512.64,Z 438.933,A -85,B 0,C 180,E1 23949.656,E2 23949.656} C_VEL
LIN {X 0,Y 512.645,Z 438.935,A -85,B 0,C 180,E1 23946.158,E2 23946.158} C_VEL
LIN {X 0,Y 512.627,Z 438.941,A -85,B 0,C 180,E1 23942.683,E2 23942.683} C_VEL
LIN {X 0,Y 512.646,Z 438.933,A -85,B 0,C 180,E1 23939.218,E2 23939.218} C_VEL
LIN {X 0,Y 512.641,Z 438.936,A -85,B 0,C 180,E1 23935.637,E2 23935.637} C_VEL
LIN {X 0,Y 512.63,Z 438.937,A -85,B 0,C 180,E1 23932.153,E2 23932.153} C_VEL
LIN {X 0,Y 512.632,Z 438.943,A -85,B 0,C 180,E1 23928.638,E2 23928.638} C_VEL
LIN {X 0,Y 512.642,Z 438.935,A -85,B 0,C 180,E1 23925.196,E2 23925.196} C_VEL
LIN {X 0,Y 512.64,Z 438.933,A -85,B 0,C 180,E1 23921.698,E2 23921.698} C_VEL
LIN {X 0,Y 512.626,Z 438.941,A -85,B 0,C 180,E1 23918.19,E2 23918.19} C_VEL
LIN {X 0,Y 512.645,Z 438.939,A -85,B 0,C 180,E1 23914.714,E2 23914.714} C_VEL
LIN {X 0,Y 512.646,Z 438.939,A -85,B 0,C 180,E1 23911.131,E2 23911.131} C_VEL
LIN {X 0,Y 512.627,Z 438.939,A -85,B 0,C 180,E1 23907.695,E2 23907.695} C_VEL
LIN {X 0,Y 512.633,Z 438.941,A -85,B 0,C 180,E1 23904.187,E2 23904.187} C_VEL
LIN {X 0,Y 512.661,Z 439.076,A -85,B 0,C 180,E1 23900.663,E2 23900.663} C_VEL
LIN {X 0,Y 517.503,Z 456.645,A -85,B 0,C 180,E1 23897.974,E2 23897.974} C_VEL
LIN {X 0,Y 516.978,Z 468.685,A -85,B 0,C 180,E1 23896.46,E2 23896.46} C_VEL
LIN {X 0,Y 515.785,Z 474.057,A -85,B 0,C 180,E1 23895.85,E2 23895.85} C_VEL
LIN {X 0,Y 509.3,Z 489.076,A -85,B 0,C 180,E1 23894.329,E2 23894.329} C_VEL
LIN {X 0,Y 508.428,Z 493.665,A -85,B 0,C 180,E1 23893.793,E2 23893.793} C_VEL
LIN {X 0,Y 507.27,Z 522.95,A -85,B 0,C 180,E1 23890.168,E2 23890.168} C_VEL
LIN {X 0,Y 506.257,Z 552.092,A -85,B 0,C 180,E1 23886.616,E2 23886.616} C_VEL
LIN {X 0,Y 506.221,Z 556.466,A -85,B 0,C 180,E1 23886.136,E2 23886.136} C_VEL
LIN {X 0,Y 508.081,Z 568.839,A -85,B 0,C 180,E1 23885.855,E2 23885.855} C_VEL
LIN {X 0,Y 507.221,Z 671.156,A -85,B 0,C 180,E1 23884.314,E2 23884.314} C_VEL
LIN {X 0,Y 507.002,Z 686.197,A -85,B 0,C 180,E1 23883.874,E2 23883.874} C_VEL
LIN {X 0,Y 506.625,Z 701.169,A -85,B 0,C 180,E1 23883.196,E2 23883.196} C_VEL
LIN {X 0,Y 506.174,Z 714.471,A -85,B 0,C 180,E1 23882.365,E2 23882.365} C_VEL
LIN {X 0,Y 505.723,Z 726.42,A -85,B 0,C 180,E1 23881.397,E2 23881.397} C_VEL
LIN {X 0,Y 505.274,Z 738.347,A -85,B 0,C 180,E1 23880.145,E2 23880.145} C_VEL
LIN {X 0,Y 504.906,Z 747.703,A -85,B 0,C 180,E1 23878.894,E2 23878.894} C_VEL
LIN {X 0,Y 504.597,Z 756.394,A -85,B 0,C 180,E1 23877.412,E2 23877.412} C_VEL
LIN {X 0,Y 504.349,Z 763.746,A -85,B 0,C 180,E1 23875.732,E2 23875.732} C_VEL
LIN {X 0,Y 504.211,Z 768.763,A -85,B 0,C 180,E1 23874.111,E2 23874.111} C_VEL
LIN {X 0,Y 504.142,Z 772.107,A -85,B 0,C 180,E1 23872.449,E2 23872.449} C_VEL
LIN {X 0,Y 504.115,Z 773.782,A -85,B 0,C 180,E1 23870.673,E2 23870.673} C_VEL
LIN {X 0,Y 504.113,Z 773.566,A -85,B 0,C 180,E1 23868.899,E2 23868.899} C_VEL
LIN {X 0,Y 504.14,Z 771.602,A -85,B 0,C 180,E1 23867.188,E2 23867.188} C_VEL
LIN {X 0,Y 504.218,Z 767.81,A -85,B 0,C 180,E1 23865.476,E2 23865.476} C_VEL
LIN {X 0,Y 504.37,Z 761.953,A -85,B 0,C 180,E1 23863.762,E2 23863.762} C_VEL
LIN {X 0,Y 504.602,Z 754.794,A -85,B 0,C 180,E1 23862.24,E2 23862.24} C_VEL
LIN {X 0,Y 504.913,Z 746.114,A -85,B 0,C 180,E1 23860.822,E2 23860.822} C_VEL
LIN {X 0,Y 505.325,Z 735.271,A -85,B 0,C 180,E1 23859.452,E2 23859.452} C_VEL
LIN {X 0,Y 505.756,Z 723.497,A -85,B 0,C 180,E1 23858.298,E2 23858.298} C_VEL
LIN {X 0,Y 506.199,Z 711.504,A -85,B 0,C 180,E1 23857.376,E2 23857.376} C_VEL
LIN {X 0,Y 506.619,Z 697.707,A -85,B 0,C 180,E1 23856.573,E2 23856.573} C_VEL
LIN {X 0,Y 506.947,Z 683.352,A -85,B 0,C 180,E1 23855.975,E2 23855.975} C_VEL
LIN {X 0,Y 507.179,Z 668.324,A -85,B 0,C 180,E1 23855.573,E2 23855.573} C_VEL
LIN {X 0,Y 507.703,Z 565.742,A -85,B 0,C 180,E1 23854.051,E2 23854.051} C_VEL
LIN {X 0,Y 506.102,Z 556.245,A -85,B 0,C 180,E1 23853.823,E2 23853.823} C_VEL
LIN {X 0,Y 506.915,Z 528.103,A -85,B 0,C 180,E1 23850.452,E2 23850.452} C_VEL
LIN {X 0,Y 507.998,Z 499.678,A -85,B 0,C 180,E1 23846.954,E2 23846.954} C_VEL
LIN {X 0,Y 509.262,Z 470.784,A -85,B 0,C 180,E1 23843.348,E2 23843.348} C_VEL
LIN {X 0,Y 509.646,Z 458.32,A -85,B 0,C 180,E1 23841.766,E2 23841.766} C_VEL
LIN {X 0,Y 504.666,Z 440.074,A -85,B 0,C 180,E1 23839.007,E2 23839.007} C_VEL
LIN {X 0,Y 504.705,Z 439.931,A -85,B 0,C 180,E1 23835.639,E2 23835.639} C_VEL
LIN {X 0,Y 504.641,Z 439.935,A -85,B 0,C 180,E1 23832.234,E2 23832.234} C_VEL
LIN {X 0,Y 504.637,Z 439.933,A -85,B 0,C 180,E1 23828.741,E2 23828.741} C_VEL
LIN {X 0,Y 504.691,Z 439.918,A -85,B 0,C 180,E1 23825.415,E2 23825.415} C_VEL
LIN {X 0,Y 504.637,Z 439.933,A -85,B 0,C 180,E1 23821.993,E2 23821.993} C_VEL
LIN {X 0,Y 504.627,Z 439.931,A -85,B 0,C 180,E1 23818.46,E2 23818.46} C_VEL
LIN {X 0,Y 504.677,Z 439.933,A -85,B 0,C 180,E1 23815.071,E2 23815.071} C_VEL
LIN {X 0,Y 504.649,Z 439.931,A -85,B 0,C 180,E1 23811.673,E2 23811.673} C_VEL
LIN {X 0,Y 504.632,Z 439.926,A -85,B 0,C 180,E1 23808.261,E2 23808.261} C_VEL
LIN {X 0,Y 504.684,Z 439.933,A -85,B 0,C 180,E1 23804.854,E2 23804.854} C_VEL
LIN {X 0,Y 504.655,Z 439.925,A -85,B 0,C 180,E1 23801.503,E2 23801.503} C_VEL
LIN {X 0,Y 504.641,Z 439.933,A -85,B 0,C 180,E1 23798.039,E2 23798.039} C_VEL
LIN {X 0,Y 504.688,Z 439.916,A -85,B 0,C 180,E1 23794.652,E2 23794.652} C_VEL
LIN {X 0,Y 504.667,Z 439.931,A -85,B 0,C 180,E1 23791.271,E2 23791.271} C_VEL
LIN {X 0,Y 504.647,Z 439.925,A -85,B 0,C 180,E1 23787.878,E2 23787.878} C_VEL
LIN {X 0,Y 504.693,Z 439.926,A -85,B 0,C 180,E1 23784.46,E2 23784.46} C_VEL
LIN {X 0,Y 504.675,Z 439.933,A -85,B 0,C 180,E1 23781.069,E2 23781.069} C_VEL
LIN {X 0,Y 504.652,Z 439.913,A -85,B 0,C 180,E1 23777.636,E2 23777.636} C_VEL
LIN {X 0,Y 504.696,Z 439.928,A -85,B 0,C 180,E1 23774.221,E2 23774.221} C_VEL
LIN {X 0,Y 504.694,Z 439.925,A -85,B 0,C 180,E1 23770.733,E2 23770.733} C_VEL
LIN {X 0,Y 504.659,Z 439.92,A -85,B 0,C 180,E1 23767.285,E2 23767.285} C_VEL
LIN {X 0,Y 504.677,Z 439.927,A -85,B 0,C 180,E1 23763.749,E2 23763.749} C_VEL
LIN {X 0,Y 504.71,Z 439.914,A -85,B 0,C 180,E1 23760.341,E2 23760.341} C_VEL
LIN {X 0,Y 504.673,Z 439.929,A -85,B 0,C 180,E1 23756.893,E2 23756.893} C_VEL
LIN {X 0,Y 504.673,Z 439.922,A -85,B 0,C 180,E1 23753.402,E2 23753.402} C_VEL
LIN {X 0,Y 504.709,Z 439.927,A -85,B 0,C 180,E1 23749.929,E2 23749.929} C_VEL
LIN {X 0,Y 504.7,Z 439.926,A -85,B 0,C 180,E1 23746.364,E2 23746.364} C_VEL
LIN {X 0,Y 504.673,Z 439.926,A -85,B 0,C 180,E1 23742.949,E2 23742.949} C_VEL
LIN {X 0,Y 504.703,Z 439.919,A -85,B 0,C 180,E1 23739.473,E2 23739.473} C_VEL
LIN {X 0,Y 504.709,Z 439.93,A -85,B 0,C 180,E1 23735.915,E2 23735.915} C_VEL
LIN {X 0,Y 504.687,Z 439.923,A -85,B 0,C 180,E1 23732.381,E2 23732.381} C_VEL
LIN {X 0,Y 504.685,Z 439.925,A -85,B 0,C 180,E1 23728.855,E2 23728.855} C_VEL
LIN {X 0,Y 504.706,Z 439.924,A -85,B 0,C 180,E1 23725.35,E2 23725.35} C_VEL
LIN {X 0,Y 504.707,Z 439.929,A -85,B 0,C 180,E1 23721.823,E2 23721.823} C_VEL
LIN {X 0,Y 504.688,Z 439.932,A -85,B 0,C 180,E1 23718.322,E2 23718.322} C_VEL
LIN {X 0,Y 504.7,Z 439.924,A -85,B 0,C 180,E1 23714.828,E2 23714.828} C_VEL
LIN {X 0,Y 504.702,Z 439.931,A -85,B 0,C 180,E1 23711.278,E2 23711.278} C_VEL
LIN {X 0,Y 504.708,Z 439.928,A -85,B 0,C 180,E1 23707.745,E2 23707.745} C_VEL
LIN {X 0,Y 504.731,Z 440.158,A -85,B 0,C 180,E1 23705.145,E2 23705.145} C_VEL
LIN {X 0,Y 511.083,Z 458.364,A -85,B 0,C 180,E1 23703.081,E2 23703.081} C_VEL
LIN {X 0,Y 512.981,Z 464.781,A -85,B 0,C 180,E1 23702.412,E2 23702.412} C_VEL
LIN {X 0,Y 511.064,Z 508.689,A -85,B 0,C 180,E1 23698.897,E2 23698.897} C_VEL
LIN {X 0,Y 509.957,Z 539.811,A -85,B 0,C 180,E1 23696.498,E2 23696.498} C_VEL
LIN {X 0,Y 511.723,Z 554.08,A -85,B 0,C 180,E1 23696.207,E2 23696.207} C_VEL
LIN {X 0,Y 510.292,Z 746.475,A -85,B 0,C 180,E1 23693.438,E2 23693.438} C_VEL
LIN {X 0,Y 509.802,Z 765.555,A -85,B 0,C 180,E1 23692.958,E2 23692.958} C_VEL
LIN {X 0,Y 509.218,Z 783.516,A -85,B 0,C 180,E1 23692.303,E2 23692.303} C_VEL
LIN {X 0,Y 508.57,Z 801.164,A -85,B 0,C 180,E1 23691.45,E2 23691.45} C_VEL
LIN {X 0,Y 507.804,Z 818.393,A -85,B 0,C 180,E1 23690.396,E2 23690.396} C_VEL
LIN {X 0,Y 507.09,Z 834.508,A -85,B 0,C 180,E1 23689.184,E2 23689.184} C_VEL
LIN {X 0,Y 506.34,Z 850.136,A -85,B 0,C 180,E1 23687.759,E2 23687.759} C_VEL
LIN {X 0,Y 505.682,Z 864.444,A -85,B 0,C 180,E1 23686.188,E2 23686.188} C_VEL
LIN {X 0,Y 505.092,Z 877.662,A -85,B 0,C 180,E1 23684.444,E2 23684.444} C_VEL
LIN {X 0,Y 504.638,Z 889.275,A -85,B 0,C 180,E1 23682.589,E2 23682.589} C_VEL
LIN {X 0,Y 504.341,Z 897.989,A -85,B 0,C 180,E1 23680.856,E2 23680.856} C_VEL
LIN {X 0,Y 504.098,Z 906.174,A -85,B 0,C 180,E1 23678.785,E2 23678.785} C_VEL
LIN {X 0,Y 503.979,Z 912.411,A -85,B 0,C 180,E1 23676.722,E2 23676.722} C_VEL
LIN {X 0,Y 503.928,Z 916.875,A -85,B 0,C 180,E1 23674.666,E2 23674.666} C_VEL
LIN {X 0,Y 503.911,Z 919.792,A -85,B 0,C 180,E1 23672.502,E2 23672.502} C_VEL
LIN {X 0,Y 503.908,Z 920.939,A -85,B 0,C 180,E1 23670.341,E2 23670.341} C_VEL
LIN {X 0,Y 503.913,Z 920.413,A -85,B 0,C 180,E1 23668.295,E2 23668.295} C_VEL
LIN {X 0,Y 503.921,Z 918.158,A -85,B 0,C 180,E1 23666.132,E2 23666.132} C_VEL
LIN {X 0,Y 503.95,Z 914.35,A -85,B 0,C 180,E1 23664.078,E2 23664.078} C_VEL
LIN {X 0,Y 504.043,Z 908.821,A -85,B 0,C 180,E1 23662.018,E2 23662.018} C_VEL
LIN {X 0,Y 504.234,Z 901.426,A -85,B 0,C 180,E1 23659.951,E2 23659.951} C_VEL
LIN {X 0,Y 504.507,Z 893.008,A -85,B 0,C 180,E1 23658.106,E2 23658.106} C_VEL
LIN {X 0,Y 504.872,Z 883.018,A -85,B 0,C 180,E1 23656.369,E2 23656.369} C_VEL
LIN {X 0,Y 505.391,Z 870.894,A -85,B 0,C 180,E1 23654.627,E2 23654.627} C_VEL
LIN {X 0,Y 506.001,Z 857.262,A -85,B 0,C 180,E1 23652.996,E2 23652.996} C_VEL
LIN {X 0,Y 506.687,Z 842.648,A -85,B 0,C 180,E1 23651.536,E2 23651.536} C_VEL
LIN {X 0,Y 507.408,Z 827.177,A -85,B 0,C 180,E1 23650.248,E2 23650.248} C_VEL
LIN {X 0,Y 508.108,Z 810.944,A -85,B 0,C 180,E1 23649.135,E2 23649.135} C_VEL
LIN {X 0,Y 508.828,Z 793.308,A -85,B 0,C 180,E1 23648.16,E2 23648.16} C_VEL
LIN {X 0,Y 509.464,Z 775.012,A -85,B 0,C 180,E1 23647.377,E2 23647.377} C_VEL
LIN {X 0,Y 510.013,Z 756.453,A -85,B 0,C 180,E1 23646.802,E2 23646.802} C_VEL
LIN {X 0,Y 510.373,Z 737.107,A -85,B 0,C 180,E1 23646.417,E2 23646.417} C_VEL
LIN {X 0,Y 511.475,Z 551.146,A -85,B 0,C 180,E1 23643.763,E2 23643.763} C_VEL
LIN {X 0,Y 509.868,Z 539.324,A -85,B 0,C 180,E1 23643.504,E2 23643.504} C_VEL
LIN {X 0,Y 511.595,Z 493.497,A -85,B 0,C 180,E1 23639.926,E2 23639.926} C_VEL
LIN {X 0,Y 512.811,Z 463.584,A -85,B 0,C 180,E1 23637.487,E2 23637.487} C_VEL
LIN {X 0,Y 505.605,Z 442.783,A -85,B 0,C 180,E1 23635.144,E2 23635.144} C_VEL
LIN {X 0,Y 504.721,Z 440.097,A -85,B 0,C 180,E1 23634.762,E2 23634.762} C_VEL
LIN {X 0,Y 504.706,Z 439.925,A -85,B 0,C 180,E1 23631.243,E2 23631.243} C_VEL
LIN {X 0,Y 504.697,Z 439.928,A -85,B 0,C 180,E1 23627.81,E2 23627.81} C_VEL
LIN {X 0,Y 504.7,Z 439.926,A -85,B 0,C 180,E1 23624.343,E2 23624.343} C_VEL
LIN {X 0,Y 504.71,Z 439.926,A -85,B 0,C 180,E1 23620.821,E2 23620.821} C_VEL
LIN {X 0,Y 504.693,Z 439.929,A -85,B 0,C 180,E1 23617.317,E2 23617.317} C_VEL
LIN {X 0,Y 504.707,Z 439.932,A -85,B 0,C 180,E1 23613.826,E2 23613.826} C_VEL
LIN {X 0,Y 504.7,Z 439.928,A -85,B 0,C 180,E1 23610.259,E2 23610.259} C_VEL
LIN {X 0,Y 504.703,Z 439.925,A -85,B 0,C 180,E1 23606.725,E2 23606.725} C_VEL
LIN {X 0,Y 504.692,Z 439.928,A -85,B 0,C 180,E1 23603.185,E2 23603.185} C_VEL
LIN {X 0,Y 504.703,Z 439.923,A -85,B 0,C 180,E1 23599.681,E2 23599.681} C_VEL
LIN {X 0,Y 504.703,Z 439.927,A -85,B 0,C 180,E1 23596.091,E2 23596.091} C_VEL
LIN {X 0,Y 504.695,Z 439.927,A -85,B 0,C 180,E1 23592.587,E2 23592.587} C_VEL
LIN {X 0,Y 504.692,Z 439.926,A -85,B 0,C 180,E1 23589.004,E2 23589.004} C_VEL
LIN {X 0,Y 504.701,Z 439.928,A -85,B 0,C 180,E1 23585.57,E2 23585.57} C_VEL
LIN {X 0,Y 504.706,Z 439.925,A -85,B 0,C 180,E1 23582.043,E2 23582.043} C_VEL
LIN {X 0,Y 504.688,Z 439.928,A -85,B 0,C 180,E1 23578.524,E2 23578.524} C_VEL
LIN {X 0,Y 504.702,Z 439.923,A -85,B 0,C 180,E1 23574.999,E2 23574.999} C_VEL
LIN {X 0,Y 504.702,Z 439.927,A -85,B 0,C 180,E1 23571.455,E2 23571.455} C_VEL
LIN {X 0,Y 504.7,Z 439.926,A -85,B 0,C 180,E1 23567.878,E2 23567.878} C_VEL
LIN {X 0,Y 504.687,Z 439.93,A -85,B 0,C 180,E1 23564.33,E2 23564.33} C_VEL
LIN {X 0,Y 504.706,Z 439.931,A -85,B 0,C 180,E1 23560.8,E2 23560.8} C_VEL
LIN {X 0,Y 504.706,Z 439.927,A -85,B 0,C 180,E1 23557.275,E2 23557.275} C_VEL
LIN {X 0,Y 504.689,Z 439.929,A -85,B 0,C 180,E1 23553.781,E2 23553.781} C_VEL
LIN {X 0,Y 504.692,Z 439.928,A -85,B 0,C 180,E1 23550.181,E2 23550.181} C_VEL
LIN {X 0,Y 504.705,Z 439.932,A -85,B 0,C 180,E1 23546.718,E2 23546.718} C_VEL
LIN {X 0,Y 504.707,Z 439.931,A -85,B 0,C 180,E1 23543.111,E2 23543.111} C_VEL
LIN {X 0,Y 504.747,Z 440.195,A -85,B 0,C 180,E1 23541.101,E2 23541.101} C_VEL
LIN {X 0,Y 509.648,Z 457.724,A -85,B 0,C 180,E1 23538.371,E2 23538.371} C_VEL
LIN {X 0,Y 510.027,Z 460.444,A -85,B 0,C 180,E1 23537.987,E2 23537.987} C_VEL
LIN {X 0,Y 508.578,Z 489.948,A -85,B 0,C 180,E1 23534.261,E2 23534.261} C_VEL
LIN {X 0,Y 508.428,Z 493.665,A -85,B 0,C 180,E1 23533.793,E2 23533.793} C_VEL
LIN {X 0,Y 507.297,Z 499.036,A -85,B 0,C 180,E1 23533.175,E2 23533.175} C_VEL
LIN {X 0,Y 500.54,Z 514.858,A -85,B 0,C 180,E1 23531.544,E2 23531.544} C_VEL
LIN {X 0,Y 499.873,Z 518.72,A -85,B 0,C 180,E1 23531.091,E2 23531.091} C_VEL
LIN {X 0,Y 498.691,Z 548.193,A -85,B 0,C 180,E1 23527.442,E2 23527.442} C_VEL
LIN {X 0,Y 498.497,Z 555.752,A -85,B 0,C 180,E1 23526.527,E2 23526.527} C_VEL
LIN {X 0,Y 499.83,Z 563.574,A -85,B 0,C 180,E1 23526.306,E2 23526.306} C_VEL
LIN {X 0,Y 500.621,Z 570.582,A -85,B 0,C 180,E1 23526.163,E2 23526.163} C_VEL
LIN {X 0,Y 499.679,Z 671.719,A -85,B 0,C 180,E1 23524.611,E2 23524.611} C_VEL
LIN {X 0,Y 499.441,Z 686.848,A -85,B 0,C 180,E1 23524.163,E2 23524.163} C_VEL
LIN {X 0,Y 499.054,Z 701.208,A -85,B 0,C 180,E1 23523.509,E2 23523.509} C_VEL
LIN {X 0,Y 498.596,Z 714.09,A -85,B 0,C 180,E1 23522.712,E2 23522.712} C_VEL
LIN {X 0,Y 498.056,Z 727.083,A -85,B 0,C 180,E1 23521.658,E2 23521.658} C_VEL
LIN {X 0,Y 497.566,Z 738.772,A -85,B 0,C 180,E1 23520.424,E2 23520.424} C_VEL
LIN {X 0,Y 497.144,Z 748.466,A -85,B 0,C 180,E1 23519.125,E2 23519.125} C_VEL
LIN {X 0,Y 496.777,Z 757.454,A -85,B 0,C 180,E1 23517.575,E2 23517.575} C_VEL
LIN {X 0,Y 496.497,Z 764.651,A -85,B 0,C 180,E1 23515.912,E2 23515.912} C_VEL
LIN {X 0,Y 496.328,Z 769.75,A -85,B 0,C 180,E1 23514.265,E2 23514.265} C_VEL
LIN {X 0,Y 496.238,Z 773.267,A -85,B 0,C 180,E1 23512.509,E2 23512.509} C_VEL
LIN {X 0,Y 496.202,Z 774.973,A -85,B 0,C 180,E1 23510.648,E2 23510.648} C_VEL
LIN {X 0,Y 496.199,Z 774.685,A -85,B 0,C 180,E1 23508.808,E2 23508.808} C_VEL
LIN {X 0,Y 496.234,Z 772.704,A -85,B 0,C 180,E1 23507.108,E2 23507.108} C_VEL
LIN {X 0,Y 496.325,Z 769.023,A -85,B 0,C 180,E1 23505.421,E2 23505.421} C_VEL
LIN {X 0,Y 496.492,Z 763.466,A -85,B 0,C 180,E1 23503.747,E2 23503.747} C_VEL
LIN {X 0,Y 496.753,Z 756.46,A -85,B 0,C 180,E1 23502.201,E2 23502.201} C_VEL
LIN {X 0,Y 497.12,Z 747.288,A -85,B 0,C 180,E1 23500.663,E2 23500.663} C_VEL
LIN {X 0,Y 497.584,Z 736.288,A -85,B 0,C 180,E1 23499.25,E2 23499.25} C_VEL
LIN {X 0,Y 498.058,Z 724.529,A -85,B 0,C 180,E1 23498.078,E2 23498.078} C_VEL
LIN {X 0,Y 498.54,Z 712.58,A -85,B 0,C 180,E1 23497.143,E2 23497.143} C_VEL
LIN {X 0,Y 498.993,Z 698.853,A -85,B 0,C 180,E1 23496.327,E2 23496.327} C_VEL
LIN {X 0,Y 499.349,Z 684.643,A -85,B 0,C 180,E1 23495.718,E2 23495.718} C_VEL
LIN {X 0,Y 499.604,Z 669.292,A -85,B 0,C 180,E1 23495.293,E2 23495.293} C_VEL
LIN {X 0,Y 500.203,Z 566.566,A -85,B 0,C 180,E1 23493.74,E2 23493.74} C_VEL
LIN {X 0,Y 498.388,Z 556.074,A -85,B 0,C 180,E1 23493.479,E2 23493.479} C_VEL
LIN {X 0,Y 499.33,Z 527.485,A -85,B 0,C 180,E1 23490,E2 23490} C_VEL
LIN {X 0,Y 500.545,Z 498.019,A -85,B 0,C 180,E1 23486.335,E2 23486.335} C_VEL
LIN {X 0,Y 501.909,Z 469.109,A -85,B 0,C 180,E1 23482.675,E2 23482.675} C_VEL
LIN {X 0,Y 502.198,Z 461.046,A -85,B 0,C 180,E1 23481.643,E2 23481.643} C_VEL
LIN {X 0,Y 497.146,Z 442.746,A -85,B 0,C 180,E1 23478.867,E2 23478.867} C_VEL
LIN {X 0,Y 496.718,Z 441.052,A -85,B 0,C 180,E1 23478.57,E2 23478.57} C_VEL
LIN {X 0,Y 496.724,Z 440.922,A -85,B 0,C 180,E1 23475.188,E2 23475.188} C_VEL
LIN {X 0,Y 496.736,Z 440.923,A -85,B 0,C 180,E1 23471.819,E2 23471.819} C_VEL
LIN {X 0,Y 496.694,Z 440.922,A -85,B 0,C 180,E1 23468.384,E2 23468.384} C_VEL
LIN {X 0,Y 496.706,Z 440.923,A -85,B 0,C 180,E1 23464.866,E2 23464.866} C_VEL
LIN {X 0,Y 496.744,Z 440.917,A -85,B 0,C 180,E1 23461.507,E2 23461.507} C_VEL
LIN {X 0,Y 496.688,Z 440.92,A -85,B 0,C 180,E1 23458.159,E2 23458.159} C_VEL
LIN {X 0,Y 496.7,Z 440.921,A -85,B 0,C 180,E1 23454.614,E2 23454.614} C_VEL
LIN {X 0,Y 496.758,Z 440.921,A -85,B 0,C 180,E1 23451.164,E2 23451.164} C_VEL
LIN {X 0,Y 496.703,Z 440.915,A -85,B 0,C 180,E1 23447.752,E2 23447.752} C_VEL
LIN {X 0,Y 496.699,Z 440.922,A -85,B 0,C 180,E1 23444.223,E2 23444.223} C_VEL
LIN {X 0,Y 496.752,Z 440.911,A -85,B 0,C 180,E1 23440.816,E2 23440.816} C_VEL
LIN {X 0,Y 496.72,Z 440.923,A -85,B 0,C 180,E1 23437.438,E2 23437.438} C_VEL
LIN {X 0,Y 496.703,Z 440.907,A -85,B 0,C 180,E1 23433.967,E2 23433.967} C_VEL
LIN {X 0,Y 496.758,Z 440.919,A -85,B 0,C 180,E1 23430.613,E2 23430.613} C_VEL
LIN {X 0,Y 496.733,Z 440.912,A -85,B 0,C 180,E1 23427.165,E2 23427.165} C_VEL
LIN {X 0,Y 496.71,Z 440.917,A -85,B 0,C 180,E1 23423.666,E2 23423.666} C_VEL
LIN {X 0,Y 496.745,Z 440.913,A -85,B 0,C 180,E1 23420.256,E2 23420.256} C_VEL
LIN {X 0,Y 496.75,Z 440.902,A -85,B 0,C 180,E1 23416.849,E2 23416.849} C_VEL
LIN {X 0,Y 496.717,Z 440.919,A -85,B 0,C 180,E1 23413.504,E2 23413.504} C_VEL
LIN {X 0,Y 496.752,Z 440.904,A -85,B 0,C 180,E1 23410.086,E2 23410.086} C_VEL
LIN {X 0,Y 496.765,Z 440.911,A -85,B 0,C 180,E1 23406.588,E2 23406.588} C_VEL
LIN {X 0,Y 496.726,Z 440.919,A -85,B 0,C 180,E1 23403.116,E2 23403.116} C_VEL
LIN {X 0,Y 496.731,Z 440.904,A -85,B 0,C 180,E1 23399.539,E2 23399.539} C_VEL
LIN {X 0,Y 496.77,Z 440.917,A -85,B 0,C 180,E1 23396.076,E2 23396.076} C_VEL
LIN {X 0,Y 496.747,Z 440.909,A -85,B 0,C 180,E1 23392.599,E2 23392.599} C_VEL
LIN {X 0,Y 496.731,Z 440.918,A -85,B 0,C 180,E1 23389.093,E2 23389.093} C_VEL
LIN {X 0,Y 496.758,Z 440.904,A -85,B 0,C 180,E1 23385.547,E2 23385.547} C_VEL
LIN {X 0,Y 496.77,Z 440.92,A -85,B 0,C 180,E1 23382.065,E2 23382.065} C_VEL
LIN {X 0,Y 496.746,Z 440.911,A -85,B 0,C 180,E1 23378.511,E2 23378.511} C_VEL
LIN {X 0,Y 496.743,Z 440.917,A -85,B 0,C 180,E1 23374.928,E2 23374.928} C_VEL
LIN {X 0,Y 496.771,Z 440.914,A -85,B 0,C 180,E1 23371.348,E2 23371.348} C_VEL
LIN {X 0,Y 496.768,Z 440.914,A -85,B 0,C 180,E1 23367.767,E2 23367.767} C_VEL
LIN {X 0,Y 496.756,Z 440.915,A -85,B 0,C 180,E1 23364.209,E2 23364.209} C_VEL
LIN {X 0,Y 496.746,Z 440.914,A -85,B 0,C 180,E1 23360.617,E2 23360.617} C_VEL
LIN {X 0,Y 496.767,Z 440.914,A -85,B 0,C 180,E1 23357.108,E2 23357.108} C_VEL
LIN {X 0,Y 496.764,Z 440.921,A -85,B 0,C 180,E1 23353.501,E2 23353.501} C_VEL
LIN {X 0,Y 496.766,Z 440.917,A -85,B 0,C 180,E1 23349.928,E2 23349.928} C_VEL
LIN {X 0,Y 496.755,Z 440.917,A -85,B 0,C 180,E1 23346.379,E2 23346.379} C_VEL
LIN {X 0,Y 496.817,Z 441.257,A -85,B 0,C 180,E1 23345.604,E2 23345.604} C_VEL
LIN {X 0,Y 505.43,Z 466.085,A -85,B 0,C 180,E1 23342.781,E2 23342.781} C_VEL
LIN {X 0,Y 505.486,Z 470.262,A -85,B 0,C 180,E1 23342.415,E2 23342.415} C_VEL
LIN {X 0,Y 503.354,Z 514.79,A -85,B 0,C 180,E1 23338.797,E2 23338.797} C_VEL
LIN {X 0,Y 502.395,Z 539.677,A -85,B 0,C 180,E1 23336.844,E2 23336.844} C_VEL
LIN {X 0,Y 504.261,Z 555.13,A -85,B 0,C 180,E1 23336.521,E2 23336.521} C_VEL
LIN {X 0,Y 502.708,Z 745.965,A -85,B 0,C 180,E1 23333.736,E2 23333.736} C_VEL
LIN {X 0,Y 502.178,Z 764.955,A -85,B 0,C 180,E1 23333.25,E2 23333.25} C_VEL
LIN {X 0,Y 501.534,Z 783.313,A -85,B 0,C 180,E1 23332.568,E2 23332.568} C_VEL
LIN {X 0,Y 500.839,Z 800.686,A -85,B 0,C 180,E1 23331.711,E2 23331.711} C_VEL
LIN {X 0,Y 500.007,Z 817.966,A -85,B 0,C 180,E1 23330.633,E2 23330.633} C_VEL
LIN {X 0,Y 499.229,Z 834.225,A -85,B 0,C 180,E1 23329.383,E2 23329.383} C_VEL
LIN {X 0,Y 498.431,Z 849.765,A -85,B 0,C 180,E1 23327.934,E2 23327.934} C_VEL
LIN {X 0,Y 497.737,Z 864.007,A -85,B 0,C 180,E1 23326.334,E2 23326.334} C_VEL
LIN {X 0,Y 497.124,Z 877.127,A -85,B 0,C 180,E1 23324.561,E2 23324.561} C_VEL
LIN {X 0,Y 496.684,Z 887.984,A -85,B 0,C 180,E1 23322.794,E2 23322.794} C_VEL
LIN {X 0,Y 496.352,Z 897.505,A -85,B 0,C 180,E1 23320.915,E2 23320.915} C_VEL
LIN {X 0,Y 496.11,Z 905.613,A -85,B 0,C 180,E1 23318.928,E2 23318.928} C_VEL
LIN {X 0,Y 495.99,Z 911.892,A -85,B 0,C 180,E1 23316.947,E2 23316.947} C_VEL
LIN {X 0,Y 495.928,Z 916.628,A -85,B 0,C 180,E1 23314.858,E2 23314.858} C_VEL
LIN {X 0,Y 495.911,Z 919.677,A -85,B 0,C 180,E1 23312.658,E2 23312.658} C_VEL
LIN {X 0,Y 495.909,Z 920.916,A -85,B 0,C 180,E1 23310.462,E2 23310.462} C_VEL
LIN {X 0,Y 495.913,Z 920.412,A -85,B 0,C 180,E1 23308.267,E2 23308.267} C_VEL
LIN {X 0,Y 495.922,Z 918.145,A -85,B 0,C 180,E1 23306.07,E2 23306.07} C_VEL
LIN {X 0,Y 495.954,Z 914.238,A -85,B 0,C 180,E1 23303.983,E2 23303.983} C_VEL
LIN {X 0,Y 496.044,Z 908.786,A -85,B 0,C 180,E1 23302.006,E2 23302.006} C_VEL
LIN {X 0,Y 496.242,Z 901.064,A -85,B 0,C 180,E1 23299.904,E2 23299.904} C_VEL
LIN {X 0,Y 496.551,Z 891.752,A -85,B 0,C 180,E1 23297.912,E2 23297.912} C_VEL
LIN {X 0,Y 496.959,Z 880.912,A -85,B 0,C 180,E1 23296.029,E2 23296.029} C_VEL
LIN {X 0,Y 497.514,Z 868.576,A -85,B 0,C 180,E1 23294.258,E2 23294.258} C_VEL
LIN {X 0,Y 498.143,Z 855.22,A -85,B 0,C 180,E1 23292.659,E2 23292.659} C_VEL
LIN {X 0,Y 498.886,Z 840.397,A -85,B 0,C 180,E1 23291.176,E2 23291.176} C_VEL
LIN {X 0,Y 499.659,Z 824.652,A -85,B 0,C 180,E1 23289.868,E2 23289.868} C_VEL
LIN {X 0,Y 500.454,Z 808.068,A -85,B 0,C 180,E1 23288.739,E2 23288.739} C_VEL
LIN {X 0,Y 501.235,Z 790.042,A -85,B 0,C 180,E1 23287.756,E2 23287.756} C_VEL
LIN {X 0,Y 501.935,Z 771.114,A -85,B 0,C 180,E1 23286.973,E2 23286.973} C_VEL
LIN {X 0,Y 502.489,Z 752.23,A -85,B 0,C 180,E1 23286.421,E2 23286.421} C_VEL
LIN {X 0,Y 502.826,Z 731.698,A -85,B 0,C 180,E1 23286.051,E2 23286.051} C_VEL
LIN {X 0,Y 504.009,Z 552.213,A -85,B 0,C 180,E1 23283.454,E2 23283.454} C_VEL
LIN {X 0,Y 502.317,Z 539.404,A -85,B 0,C 180,E1 23283.168,E2 23283.168} C_VEL
LIN {X 0,Y 504.226,Z 494.166,A -85,B 0,C 180,E1 23279.563,E2 23279.563} C_VEL
LIN {X 0,Y 505.576,Z 466.53,A -85,B 0,C 180,E1 23277.267,E2 23277.267} C_VEL
LIN {X 0,Y 498.915,Z 447.054,A -85,B 0,C 180,E1 23275.029,E2 23275.029} C_VEL
LIN {X 0,Y 496.795,Z 441.123,A -85,B 0,C 180,E1 23274.251,E2 23274.251} C_VEL
LIN {X 0,Y 496.76,Z 440.917,A -85,B 0,C 180,E1 23270.797,E2 23270.797} C_VEL
LIN {X 0,Y 496.761,Z 440.913,A -85,B 0,C 180,E1 23267.278,E2 23267.278} C_VEL
LIN {X 0,Y 496.757,Z 440.921,A -85,B 0,C 180,E1 23263.66,E2 23263.66} C_VEL
LIN {X 0,Y 496.767,Z 440.919,A -85,B 0,C 180,E1 23260.096,E2 23260.096} C_VEL
LIN {X 0,Y 496.763,Z 440.916,A -85,B 0,C 180,E1 23256.568,E2 23256.568} C_VEL
LIN {X 0,Y 496.757,Z 440.913,A -85,B 0,C 180,E1 23253.056,E2 23253.056} C_VEL
LIN {X 0,Y 496.757,Z 440.915,A -85,B 0,C 180,E1 23249.414,E2 23249.414} C_VEL
LIN {X 0,Y 496.765,Z 440.92,A -85,B 0,C 180,E1 23245.882,E2 23245.882} C_VEL
LIN {X 0,Y 496.764,Z 440.914,A -85,B 0,C 180,E1 23242.234,E2 23242.234} C_VEL
LIN {X 0,Y 496.758,Z 440.911,A -85,B 0,C 180,E1 23238.665,E2 23238.665} C_VEL
LIN {X 0,Y 496.753,Z 440.908,A -85,B 0,C 180,E1 23235.049,E2 23235.049} C_VEL
LIN {X 0,Y 496.765,Z 440.921,A -85,B 0,C 180,E1 23231.494,E2 23231.494} C_VEL
LIN {X 0,Y 496.765,Z 440.914,A -85,B 0,C 180,E1 23227.866,E2 23227.866} C_VEL
LIN {X 0,Y 496.755,Z 440.907,A -85,B 0,C 180,E1 23224.386,E2 23224.386} C_VEL
LIN {X 0,Y 496.752,Z 440.912,A -85,B 0,C 180,E1 23220.807,E2 23220.807} C_VEL
LIN {X 0,Y 496.765,Z 440.921,A -85,B 0,C 180,E1 23217.231,E2 23217.231} C_VEL
LIN {X 0,Y 496.766,Z 440.912,A -85,B 0,C 180,E1 23213.644,E2 23213.644} C_VEL
LIN {X 0,Y 496.751,Z 440.91,A -85,B 0,C 180,E1 23210.149,E2 23210.149} C_VEL
LIN {X 0,Y 496.756,Z 440.911,A -85,B 0,C 180,E1 23206.616,E2 23206.616} C_VEL
LIN {X 0,Y 496.765,Z 440.918,A -85,B 0,C 180,E1 23203.152,E2 23203.152} C_VEL
LIN {X 0,Y 496.765,Z 440.914,A -85,B 0,C 180,E1 23199.622,E2 23199.622} C_VEL
LIN {X 0,Y 496.749,Z 440.914,A -85,B 0,C 180,E1 23196.135,E2 23196.135} C_VEL
LIN {X 0,Y 496.768,Z 440.915,A -85,B 0,C 180,E1 23192.554,E2 23192.554} C_VEL
LIN {X 0,Y 496.767,Z 440.918,A -85,B 0,C 180,E1 23188.985,E2 23188.985} C_VEL
LIN {X 0,Y 496.759,Z 440.917,A -85,B 0,C 180,E1 23185.408,E2 23185.408} C_VEL
LIN {X 0,Y 496.746,Z 440.922,A -85,B 0,C 180,E1 23181.834,E2 23181.834} C_VEL
LIN {X 0,Y 496.841,Z 441.493,A -85,B 0,C 180,E1 23181.549,E2 23181.549} C_VEL
LIN {X 0,Y 501.682,Z 458.237,A -85,B 0,C 180,E1 23178.875,E2 23178.875} C_VEL
LIN {X 0,Y 502.6,Z 462.715,A -85,B 0,C 180,E1 23178.207,E2 23178.207} C_VEL
LIN {X 0,Y 501.027,Z 491.904,A -85,B 0,C 180,E1 23174.464,E2 23174.464} C_VEL
LIN {X 0,Y 499.873,Z 518.72,A -85,B 0,C 180,E1 23171.091,E2 23171.091} C_VEL
LIN {X 0,Y 498.718,Z 524.137,A -85,B 0,C 180,E1 23170.467,E2 23170.467} C_VEL
LIN {X 0,Y 491.931,Z 539.958,A -85,B 0,C 180,E1 23168.81,E2 23168.81} C_VEL
LIN {X 0,Y 491.249,Z 543.822,A -85,B 0,C 180,E1 23168.351,E2 23168.351} C_VEL
LIN {X 0,Y 490.844,Z 555.902,A -85,B 0,C 180,E1 23166.88,E2 23166.88} C_VEL
LIN {X 0,Y 493.2,Z 570.551,A -85,B 0,C 180,E1 23166.51,E2 23166.51} C_VEL
LIN {X 0,Y 492.153,Z 672.411,A -85,B 0,C 180,E1 23164.916,E2 23164.916} C_VEL
LIN {X 0,Y 491.893,Z 687.683,A -85,B 0,C 180,E1 23164.454,E2 23164.454} C_VEL
LIN {X 0,Y 491.485,Z 701.699,A -85,B 0,C 180,E1 23163.807,E2 23163.807} C_VEL
LIN {X 0,Y 490.968,Z 715.195,A -85,B 0,C 180,E1 23162.96,E2 23162.96} C_VEL
LIN {X 0,Y 490.377,Z 728.301,A -85,B 0,C 180,E1 23161.876,E2 23161.876} C_VEL
LIN {X 0,Y 489.845,Z 739.804,A -85,B 0,C 180,E1 23160.639,E2 23160.639} C_VEL
LIN {X 0,Y 489.391,Z 749.234,A -85,B 0,C 180,E1 23159.362,E2 23159.362} C_VEL
LIN {X 0,Y 488.971,Z 758.289,A -85,B 0,C 180,E1 23157.789,E2 23157.789} C_VEL
LIN {X 0,Y 488.665,Z 765.072,A -85,B 0,C 180,E1 23156.229,E2 23156.229} C_VEL
LIN {X 0,Y 488.463,Z 770.422,A -85,B 0,C 180,E1 23154.553,E2 23154.553} C_VEL
LIN {X 0,Y 488.344,Z 774.131,A -85,B 0,C 180,E1 23152.766,E2 23152.766} C_VEL
LIN {X 0,Y 488.29,Z 775.978,A -85,B 0,C 180,E1 23150.973,E2 23150.973} C_VEL
LIN {X 0,Y 488.284,Z 776.114,A -85,B 0,C 180,E1 23149.249,E2 23149.249} C_VEL
LIN {X 0,Y 488.316,Z 774.385,A -85,B 0,C 180,E1 23147.394,E2 23147.394} C_VEL
LIN {X 0,Y 488.406,Z 771.028,A -85,B 0,C 180,E1 23145.678,E2 23145.678} C_VEL
LIN {X 0,Y 488.586,Z 765.901,A -85,B 0,C 180,E1 23143.974,E2 23143.974} C_VEL
LIN {X 0,Y 488.875,Z 758.71,A -85,B 0,C 180,E1 23142.281,E2 23142.281} C_VEL
LIN {X 0,Y 489.227,Z 750.63,A -85,B 0,C 180,E1 23140.837,E2 23140.837} C_VEL
LIN {X 0,Y 489.668,Z 741.229,A -85,B 0,C 180,E1 23139.512,E2 23139.512} C_VEL
LIN {X 0,Y 490.183,Z 729.995,A -85,B 0,C 180,E1 23138.268,E2 23138.268} C_VEL
LIN {X 0,Y 490.715,Z 717.691,A -85,B 0,C 180,E1 23137.198,E2 23137.198} C_VEL
LIN {X 0,Y 491.234,Z 704.343,A -85,B 0,C 180,E1 23136.31,E2 23136.31} C_VEL
LIN {X 0,Y 491.652,Z 690.509,A -85,B 0,C 180,E1 23135.631,E2 23135.631} C_VEL
LIN {X 0,Y 491.969,Z 675.494,A -85,B 0,C 180,E1 23135.127,E2 23135.127} C_VEL
LIN {X 0,Y 492.176,Z 654.276,A -85,B 0,C 180,E1 23134.743,E2 23134.743} C_VEL
LIN {X 0,Y 492.738,Z 567.605,A -85,B 0,C 180,E1 23133.423,E2 23133.423} C_VEL
LIN {X 0,Y 490.675,Z 555.871,A -85,B 0,C 180,E1 23133.124,E2 23133.124} C_VEL
LIN {X 0,Y 491.726,Z 526.783,A -85,B 0,C 180,E1 23129.534,E2 23129.534} C_VEL
LIN {X 0,Y 493.018,Z 498.189,A -85,B 0,C 180,E1 23125.929,E2 23125.929} C_VEL
LIN {X 0,Y 494.483,Z 469.175,A -85,B 0,C 180,E1 23122.214,E2 23122.214} C_VEL
LIN {X 0,Y 494.566,Z 462.988,A -85,B 0,C 180,E1 23121.396,E2 23121.396} C_VEL
LIN {X 0,Y 489.393,Z 444.242,A -85,B 0,C 180,E1 23118.51,E2 23118.51} C_VEL
LIN {X 0,Y 488.798,Z 442.012,A -85,B 0,C 180,E1 23118.107,E2 23118.107} C_VEL
LIN {X 0,Y 488.76,Z 441.914,A -85,B 0,C 180,E1 23114.698,E2 23114.698} C_VEL
LIN {X 0,Y 488.798,Z 441.909,A -85,B 0,C 180,E1 23111.267,E2 23111.267} C_VEL
LIN {X 0,Y 488.779,Z 441.901,A -85,B 0,C 180,E1 23107.889,E2 23107.889} C_VEL
LIN {X 0,Y 488.752,Z 441.911,A -85,B 0,C 180,E1 23104.427,E2 23104.427} C_VEL
LIN {X 0,Y 488.781,Z 441.913,A -85,B 0,C 180,E1 23101,E2 23101} C_VEL
LIN {X 0,Y 488.784,Z 441.906,A -85,B 0,C 180,E1 23097.591,E2 23097.591} C_VEL
LIN {X 0,Y 488.751,Z 441.91,A -85,B 0,C 180,E1 23094.191,E2 23094.191} C_VEL
LIN {X 0,Y 488.773,Z 441.912,A -85,B 0,C 180,E1 23090.648,E2 23090.648} C_VEL
LIN {X 0,Y 488.808,Z 441.9,A -85,B 0,C 180,E1 23087.226,E2 23087.226} C_VEL
LIN {X 0,Y 488.763,Z 441.912,A -85,B 0,C 180,E1 23083.769,E2 23083.769} C_VEL
LIN {X 0,Y 488.768,Z 441.905,A -85,B 0,C 180,E1 23080.267,E2 23080.267} C_VEL
LIN {X 0,Y 488.822,Z 441.906,A -85,B 0,C 180,E1 23076.891,E2 23076.891} C_VEL
LIN {X 0,Y 488.781,Z 441.896,A -85,B 0,C 180,E1 23073.386,E2 23073.386} C_VEL
LIN {X 0,Y 488.77,Z 441.91,A -85,B 0,C 180,E1 23069.944,E2 23069.944} C_VEL
LIN {X 0,Y 488.822,Z 441.889,A -85,B 0,C 180,E1 23066.613,E2 23066.613} C_VEL
LIN {X 0,Y 488.794,Z 441.907,A -85,B 0,C 180,E1 23063.126,E2 23063.126} C_VEL
LIN {X 0,Y 488.775,Z 441.904,A -85,B 0,C 180,E1 23059.602,E2 23059.602} C_VEL
LIN {X 0,Y 488.805,Z 441.9,A -85,B 0,C 180,E1 23056.153,E2 23056.153} C_VEL
LIN {X 0,Y 488.824,Z 441.91,A -85,B 0,C 180,E1 23052.663,E2 23052.663} C_VEL
LIN {X 0,Y 488.784,Z 441.895,A -85,B 0,C 180,E1 23049.181,E2 23049.181} C_VEL
LIN {X 0,Y 488.787,Z 441.905,A -85,B 0,C 180,E1 23045.517,E2 23045.517} C_VEL
LIN {X 0,Y 488.821,Z 441.895,A -85,B 0,C 180,E1 23041.993,E2 23041.993} C_VEL
LIN {X 0,Y 488.825,Z 441.897,A -85,B 0,C 180,E1 23038.477,E2 23038.477} C_VEL
LIN {X 0,Y 488.793,Z 441.909,A -85,B 0,C 180,E1 23034.954,E2 23034.954} C_VEL
LIN {X 0,Y 488.794,Z 441.895,A -85,B 0,C 180,E1 23031.294,E2 23031.294} C_VEL
LIN {X 0,Y 488.83,Z 441.904,A -85,B 0,C 180,E1 23027.838,E2 23027.838} C_VEL
LIN {X 0,Y 488.83,Z 441.896,A -85,B 0,C 180,E1 23024.215,E2 23024.215} C_VEL
LIN {X 0,Y 488.804,Z 441.909,A -85,B 0,C 180,E1 23020.648,E2 23020.648} C_VEL
LIN {X 0,Y 488.804,Z 441.902,A -85,B 0,C 180,E1 23016.998,E2 23016.998} C_VEL
LIN {X 0,Y 488.829,Z 441.894,A -85,B 0,C 180,E1 23013.519,E2 23013.519} C_VEL
LIN {X 0,Y 488.834,Z 441.906,A -85,B 0,C 180,E1 23009.906,E2 23009.906} C_VEL
LIN {X 0,Y 488.813,Z 441.908,A -85,B 0,C 180,E1 23006.336,E2 23006.336} C_VEL
LIN {X 0,Y 488.809,Z 441.906,A -85,B 0,C 180,E1 23002.722,E2 23002.722} C_VEL
LIN {X 0,Y 488.833,Z 441.904,A -85,B 0,C 180,E1 22999.116,E2 22999.116} C_VEL
LIN {X 0,Y 488.826,Z 441.906,A -85,B 0,C 180,E1 22995.55,E2 22995.55} C_VEL
LIN {X 0,Y 488.821,Z 441.906,A -85,B 0,C 180,E1 22991.98,E2 22991.98} C_VEL
LIN {X 0,Y 488.816,Z 441.908,A -85,B 0,C 180,E1 22988.426,E2 22988.426} C_VEL
LIN {X 0,Y 488.855,Z 442.178,A -85,B 0,C 180,E1 22986.122,E2 22986.122} C_VEL
LIN {X 0,Y 495.939,Z 462.364,A -85,B 0,C 180,E1 22983.733,E2 22983.733} C_VEL
LIN {X 0,Y 498.323,Z 469.512,A -85,B 0,C 180,E1 22982.939,E2 22982.939} C_VEL
LIN {X 0,Y 495.938,Z 514.739,A -85,B 0,C 180,E1 22979.195,E2 22979.195} C_VEL
LIN {X 0,Y 494.859,Z 539.554,A -85,B 0,C 180,E1 22977.203,E2 22977.203} C_VEL
LIN {X 0,Y 496.814,Z 556.078,A -85,B 0,C 180,E1 22976.846,E2 22976.846} C_VEL
LIN {X 0,Y 495.14,Z 745.286,A -85,B 0,C 180,E1 22974.046,E2 22974.046} C_VEL
LIN {X 0,Y 494.579,Z 764.227,A -85,B 0,C 180,E1 22973.556,E2 22973.556} C_VEL
LIN {X 0,Y 493.897,Z 782.381,A -85,B 0,C 180,E1 22972.873,E2 22972.873} C_VEL
LIN {X 0,Y 493.106,Z 800.432,A -85,B 0,C 180,E1 22971.967,E2 22971.967} C_VEL
LIN {X 0,Y 492.208,Z 817.738,A -85,B 0,C 180,E1 22970.864,E2 22970.864} C_VEL
LIN {X 0,Y 491.374,Z 833.934,A -85,B 0,C 180,E1 22969.589,E2 22969.589} C_VEL
LIN {X 0,Y 490.526,Z 849.383,A -85,B 0,C 180,E1 22968.115,E2 22968.115} C_VEL
LIN {X 0,Y 489.794,Z 863.563,A -85,B 0,C 180,E1 22966.485,E2 22966.485} C_VEL
LIN {X 0,Y 489.196,Z 875.782,A -85,B 0,C 180,E1 22964.803,E2 22964.803} C_VEL
LIN {X 0,Y 488.732,Z 886.69,A -85,B 0,C 180,E1 22963.005,E2 22963.005} C_VEL
LIN {X 0,Y 488.391,Z 896.251,A -85,B 0,C 180,E1 22961.096,E2 22961.096} C_VEL
LIN {X 0,Y 488.153,Z 904.392,A -85,B 0,C 180,E1 22959.075,E2 22959.075} C_VEL
LIN {X 0,Y 488.035,Z 911.02,A -85,B 0,C 180,E1 22956.943,E2 22956.943} C_VEL
LIN {X 0,Y 487.98,Z 915.767,A -85,B 0,C 180,E1 22954.819,E2 22954.819} C_VEL
LIN {X 0,Y 487.959,Z 918.749,A -85,B 0,C 180,E1 22952.701,E2 22952.701} C_VEL
LIN {X 0,Y 487.956,Z 920.042,A -85,B 0,C 180,E1 22950.587,E2 22950.587} C_VEL
LIN {X 0,Y 487.959,Z 919.6,A -85,B 0,C 180,E1 22948.356,E2 22948.356} C_VEL
LIN {X 0,Y 487.973,Z 917.294,A -85,B 0,C 180,E1 22946.123,E2 22946.123} C_VEL
LIN {X 0,Y 488.007,Z 913.336,A -85,B 0,C 180,E1 22944.002,E2 22944.002} C_VEL
LIN {X 0,Y 488.091,Z 907.55,A -85,B 0,C 180,E1 22941.874,E2 22941.874} C_VEL
LIN {X 0,Y 488.283,Z 899.79,A -85,B 0,C 180,E1 22939.738,E2 22939.738} C_VEL
LIN {X 0,Y 488.595,Z 890.434,A -85,B 0,C 180,E1 22937.712,E2 22937.712} C_VEL
LIN {X 0,Y 489.018,Z 879.541,A -85,B 0,C 180,E1 22935.797,E2 22935.797} C_VEL
LIN {X 0,Y 489.602,Z 867.136,A -85,B 0,C 180,E1 22933.997,E2 22933.997} C_VEL
LIN {X 0,Y 490.308,Z 853.168,A -85,B 0,C 180,E1 22932.311,E2 22932.311} C_VEL
LIN {X 0,Y 491.113,Z 838.203,A -85,B 0,C 180,E1 22930.811,E2 22930.811} C_VEL
LIN {X 0,Y 491.948,Z 822.106,A -85,B 0,C 180,E1 22929.476,E2 22929.476} C_VEL
LIN {X 0,Y 492.843,Z 804.669,A -85,B 0,C 180,E1 22928.306,E2 22928.306} C_VEL
LIN {X 0,Y 493.631,Z 787.066,A -85,B 0,C 180,E1 22927.366,E2 22927.366} C_VEL
LIN {X 0,Y 494.363,Z 768.781,A -85,B 0,C 180,E1 22926.622,E2 22926.622} C_VEL
LIN {X 0,Y 494.947,Z 750.144,A -85,B 0,C 180,E1 22926.087,E2 22926.087} C_VEL
LIN {X 0,Y 495.284,Z 727.774,A -85,B 0,C 180,E1 22925.696,E2 22925.696} C_VEL
LIN {X 0,Y 496.544,Z 553.171,A -85,B 0,C 180,E1 22923.131,E2 22923.131} C_VEL
LIN {X 0,Y 494.808,Z 539.712,A -85,B 0,C 180,E1 22922.827,E2 22922.827} C_VEL
LIN {X 0,Y 496.876,Z 495.489,A -85,B 0,C 180,E1 22919.232,E2 22919.232} C_VEL
LIN {X 0,Y 498.289,Z 469.243,A -85,B 0,C 180,E1 22917.008,E2 22917.008} C_VEL
LIN {X 0,Y 491.585,Z 449.814,A -85,B 0,C 180,E1 22914.715,E2 22914.715} C_VEL
LIN {X 0,Y 488.846,Z 442.113,A -85,B 0,C 180,E1 22913.692,E2 22913.692} C_VEL
LIN {X 0,Y 488.831,Z 441.909,A -85,B 0,C 180,E1 22910.192,E2 22910.192} C_VEL
LIN {X 0,Y 488.822,Z 441.904,A -85,B 0,C 180,E1 22906.563,E2 22906.563} C_VEL
LIN {X 0,Y 488.827,Z 441.905,A -85,B 0,C 180,E1 22902.924,E2 22902.924} C_VEL
LIN {X 0,Y 488.816,Z 441.901,A -85,B 0,C 180,E1 22899.353,E2 22899.353} C_VEL
LIN {X 0,Y 488.825,Z 441.902,A -85,B 0,C 180,E1 22895.802,E2 22895.802} C_VEL
LIN {X 0,Y 488.823,Z 441.901,A -85,B 0,C 180,E1 22892.266,E2 22892.266} C_VEL
LIN {X 0,Y 488.831,Z 441.898,A -85,B 0,C 180,E1 22888.66,E2 22888.66} C_VEL
LIN {X 0,Y 488.815,Z 441.901,A -85,B 0,C 180,E1 22885.022,E2 22885.022} C_VEL
LIN {X 0,Y 488.827,Z 441.909,A -85,B 0,C 180,E1 22881.461,E2 22881.461} C_VEL
LIN {X 0,Y 488.824,Z 441.903,A -85,B 0,C 180,E1 22877.867,E2 22877.867} C_VEL
LIN {X 0,Y 488.829,Z 441.891,A -85,B 0,C 180,E1 22874.208,E2 22874.208} C_VEL
LIN {X 0,Y 488.814,Z 441.899,A -85,B 0,C 180,E1 22870.608,E2 22870.608} C_VEL
LIN {X 0,Y 488.814,Z 441.908,A -85,B 0,C 180,E1 22866.931,E2 22866.931} C_VEL
LIN {X 0,Y 488.826,Z 441.9,A -85,B 0,C 180,E1 22863.4,E2 22863.4} C_VEL
LIN {X 0,Y 488.827,Z 441.895,A -85,B 0,C 180,E1 22859.765,E2 22859.765} C_VEL
LIN {X 0,Y 488.818,Z 441.902,A -85,B 0,C 180,E1 22856.129,E2 22856.129} C_VEL
LIN {X 0,Y 488.812,Z 441.908,A -85,B 0,C 180,E1 22852.596,E2 22852.596} C_VEL
LIN {X 0,Y 488.827,Z 441.904,A -85,B 0,C 180,E1 22849.034,E2 22849.034} C_VEL
LIN {X 0,Y 488.827,Z 441.898,A -85,B 0,C 180,E1 22845.428,E2 22845.428} C_VEL
LIN {X 0,Y 488.816,Z 441.901,A -85,B 0,C 180,E1 22841.886,E2 22841.886} C_VEL
LIN {X 0,Y 488.811,Z 441.907,A -85,B 0,C 180,E1 22838.225,E2 22838.225} C_VEL
LIN {X 0,Y 488.828,Z 441.905,A -85,B 0,C 180,E1 22834.691,E2 22834.691} C_VEL
LIN {X 0,Y 488.83,Z 441.907,A -85,B 0,C 180,E1 22831.096,E2 22831.096} C_VEL
LIN {X 0,Y 488.815,Z 441.905,A -85,B 0,C 180,E1 22827.594,E2 22827.594} C_VEL
LIN {X 0,Y 488.811,Z 441.907,A -85,B 0,C 180,E1 22824.051,E2 22824.051} C_VEL
LIN {X 0,Y 488.856,Z 442.187,A -85,B 0,C 180,E1 22822.128,E2 22822.128} C_VEL
LIN {X 0,Y 493.85,Z 459.299,A -85,B 0,C 180,E1 22819.312,E2 22819.312} C_VEL
LIN {X 0,Y 495.163,Z 465.517,A -85,B 0,C 180,E1 22818.368,E2 22818.368} C_VEL
LIN {X 0,Y 493.506,Z 493.976,A -85,B 0,C 180,E1 22814.671,E2 22814.671} C_VEL
LIN {X 0,Y 492.15,Z 522.663,A -85,B 0,C 180,E1 22811.011,E2 22811.011} C_VEL
LIN {X 0,Y 491.249,Z 543.822,A -85,B 0,C 180,E1 22808.351,E2 22808.351} C_VEL
LIN {X 0,Y 490.179,Z 547.694,A -85,B 0,C 180,E1 22807.932,E2 22807.932} C_VEL
LIN {X 0,Y 486.775,Z 554.295,A -85,B 0,C 180,E1 22807.431,E2 22807.431} C_VEL
LIN {X 0,Y 484.84,Z 559.649,A -85,B 0,C 180,E1 22807.169,E2 22807.169} C_VEL
LIN {X 0,Y 484.694,Z 563.985,A -85,B 0,C 180,E1 22807.03,E2 22807.03} C_VEL
LIN {X 0,Y 485.79,Z 572.02,A -85,B 0,C 180,E1 22806.847,E2 22806.847} C_VEL
LIN {X 0,Y 484.661,Z 672.843,A -85,B 0,C 180,E1 22805.241,E2 22805.241} C_VEL
LIN {X 0,Y 484.373,Z 688.575,A -85,B 0,C 180,E1 22804.757,E2 22804.757} C_VEL
LIN {X 0,Y 483.901,Z 703.522,A -85,B 0,C 180,E1 22804.048,E2 22804.048} C_VEL
LIN {X 0,Y 483.336,Z 716.833,A -85,B 0,C 180,E1 22803.182,E2 22803.182} C_VEL
LIN {X 0,Y 482.707,Z 729.658,A -85,B 0,C 180,E1 22802.092,E2 22802.092} C_VEL
LIN {X 0,Y 482.09,Z 741.815,A -85,B 0,C 180,E1 22800.746,E2 22800.746} C_VEL
LIN {X 0,Y 481.555,Z 751.683,A -85,B 0,C 180,E1 22799.341,E2 22799.341} C_VEL
LIN {X 0,Y 481.142,Z 759.782,A -85,B 0,C 180,E1 22797.877,E2 22797.877} C_VEL
LIN {X 0,Y 480.785,Z 766.953,A -85,B 0,C 180,E1 22796.16,E2 22796.16} C_VEL
LIN {X 0,Y 480.56,Z 772.045,A -85,B 0,C 180,E1 22794.459,E2 22794.459} C_VEL
LIN {X 0,Y 480.433,Z 775.573,A -85,B 0,C 180,E1 22792.644,E2 22792.644} C_VEL
LIN {X 0,Y 480.375,Z 777.29,A -85,B 0,C 180,E1 22790.722,E2 22790.722} C_VEL
LIN {X 0,Y 480.37,Z 777.114,A -85,B 0,C 180,E1 22788.947,E2 22788.947} C_VEL
LIN {X 0,Y 480.417,Z 775.328,A -85,B 0,C 180,E1 22787.189,E2 22787.189} C_VEL
LIN {X 0,Y 480.539,Z 771.49,A -85,B 0,C 180,E1 22785.322,E2 22785.322} C_VEL
LIN {X 0,Y 480.755,Z 766.037,A -85,B 0,C 180,E1 22783.592,E2 22783.592} C_VEL
LIN {X 0,Y 481.079,Z 759.163,A -85,B 0,C 180,E1 22781.995,E2 22781.995} C_VEL
LIN {X 0,Y 481.517,Z 750.115,A -85,B 0,C 180,E1 22780.408,E2 22780.408} C_VEL
LIN {X 0,Y 482.017,Z 740.347,A -85,B 0,C 180,E1 22779.07,E2 22779.07} C_VEL
LIN {X 0,Y 482.604,Z 728.571,A -85,B 0,C 180,E1 22777.799,E2 22777.799} C_VEL
LIN {X 0,Y 483.223,Z 715.157,A -85,B 0,C 180,E1 22776.687,E2 22776.687} C_VEL
LIN {X 0,Y 483.727,Z 702.232,A -85,B 0,C 180,E1 22775.872,E2 22775.872} C_VEL
LIN {X 0,Y 484.165,Z 688.095,A -85,B 0,C 180,E1 22775.213,E2 22775.213} C_VEL
LIN {X 0,Y 484.464,Z 672.318,A -85,B 0,C 180,E1 22774.735,E2 22774.735} C_VEL
LIN {X 0,Y 485.255,Z 568.62,A -85,B 0,C 180,E1 22773.1,E2 22773.1} C_VEL
LIN {X 0,Y 482.995,Z 556.046,A -85,B 0,C 180,E1 22772.788,E2 22772.788} C_VEL
LIN {X 0,Y 483.214,Z 548.549,A -85,B 0,C 180,E1 22771.897,E2 22771.897} C_VEL
LIN {X 0,Y 484.483,Z 518.642,A -85,B 0,C 180,E1 22768.108,E2 22768.108} C_VEL
LIN {X 0,Y 485.931,Z 490.131,A -85,B 0,C 180,E1 22764.45,E2 22764.45} C_VEL
LIN {X 0,Y 487.233,Z 466.152,A -85,B 0,C 180,E1 22761.325,E2 22761.325} C_VEL
LIN {X 0,Y 482.062,Z 447.336,A -85,B 0,C 180,E1 22758.393,E2 22758.393} C_VEL
LIN {X 0,Y 480.892,Z 442.98,A -85,B 0,C 180,E1 22757.634,E2 22757.634} C_VEL
LIN {X 0,Y 480.832,Z 442.903,A -85,B 0,C 180,E1 22754.192,E2 22754.192} C_VEL
LIN {X 0,Y 480.819,Z 442.899,A -85,B 0,C 180,E1 22750.692,E2 22750.692} C_VEL
LIN {X 0,Y 480.859,Z 442.875,A -85,B 0,C 180,E1 22747.247,E2 22747.247} C_VEL
LIN {X 0,Y 480.848,Z 442.9,A -85,B 0,C 180,E1 22743.71,E2 22743.71} C_VEL
LIN {X 0,Y 480.81,Z 442.902,A -85,B 0,C 180,E1 22740.335,E2 22740.335} C_VEL
LIN {X 0,Y 480.835,Z 442.901,A -85,B 0,C 180,E1 22736.846,E2 22736.846} C_VEL
LIN {X 0,Y 480.863,Z 442.892,A -85,B 0,C 180,E1 22733.361,E2 22733.361} C_VEL
LIN {X 0,Y 480.818,Z 442.902,A -85,B 0,C 180,E1 22729.93,E2 22729.93} C_VEL
LIN {X 0,Y 480.824,Z 442.897,A -85,B 0,C 180,E1 22726.339,E2 22726.339} C_VEL
LIN {X 0,Y 480.868,Z 442.889,A -85,B 0,C 180,E1 22722.838,E2 22722.838} C_VEL
LIN {X 0,Y 480.837,Z 442.895,A -85,B 0,C 180,E1 22719.514,E2 22719.514} C_VEL
LIN {X 0,Y 480.825,Z 442.894,A -85,B 0,C 180,E1 22716.01,E2 22716.01} C_VEL
LIN {X 0,Y 480.87,Z 442.894,A -85,B 0,C 180,E1 22712.584,E2 22712.584} C_VEL
LIN {X 0,Y 480.863,Z 442.9,A -85,B 0,C 180,E1 22709.115,E2 22709.115} C_VEL
LIN {X 0,Y 480.831,Z 442.881,A -85,B 0,C 180,E1 22705.628,E2 22705.628} C_VEL
LIN {X 0,Y 480.851,Z 442.897,A -85,B 0,C 180,E1 22702.109,E2 22702.109} C_VEL
LIN {X 0,Y 480.887,Z 442.878,A -85,B 0,C 180,E1 22698.675,E2 22698.675} C_VEL
LIN {X 0,Y 480.847,Z 442.891,A -85,B 0,C 180,E1 22695.189,E2 22695.189} C_VEL
LIN {X 0,Y 480.844,Z 442.894,A -85,B 0,C 180,E1 22691.637,E2 22691.637} C_VEL
LIN {X 0,Y 480.883,Z 442.879,A -85,B 0,C 180,E1 22688.128,E2 22688.128} C_VEL
LIN {X 0,Y 480.886,Z 442.899,A -85,B 0,C 180,E1 22684.532,E2 22684.532} C_VEL
LIN {X 0,Y 480.854,Z 442.887,A -85,B 0,C 180,E1 22680.953,E2 22680.953} C_VEL
LIN {X 0,Y 480.853,Z 442.894,A -85,B 0,C 180,E1 22677.378,E2 22677.378} C_VEL
LIN {X 0,Y 480.884,Z 442.885,A -85,B 0,C 180,E1 22673.793,E2 22673.793} C_VEL
LIN {X 0,Y 480.891,Z 442.891,A -85,B 0,C 180,E1 22670.184,E2 22670.184} C_VEL
LIN {X 0,Y 480.865,Z 442.897,A -85,B 0,C 180,E1 22666.656,E2 22666.656} C_VEL
LIN {X 0,Y 480.859,Z 442.892,A -85,B 0,C 180,E1 22663.037,E2 22663.037} C_VEL
LIN {X 0,Y 480.882,Z 442.885,A -85,B 0,C 180,E1 22659.428,E2 22659.428} C_VEL
LIN {X 0,Y 480.892,Z 442.896,A -85,B 0,C 180,E1 22655.821,E2 22655.821} C_VEL
LIN {X 0,Y 480.88,Z 442.888,A -85,B 0,C 180,E1 22652.242,E2 22652.242} C_VEL
LIN {X 0,Y 480.866,Z 442.893,A -85,B 0,C 180,E1 22648.68,E2 22648.68} C_VEL
LIN {X 0,Y 480.883,Z 442.891,A -85,B 0,C 180,E1 22645.125,E2 22645.125} C_VEL
LIN {X 0,Y 480.888,Z 442.892,A -85,B 0,C 180,E1 22641.561,E2 22641.561} C_VEL
LIN {X 0,Y 480.888,Z 442.894,A -85,B 0,C 180,E1 22637.926,E2 22637.926} C_VEL
LIN {X 0,Y 480.874,Z 442.893,A -85,B 0,C 180,E1 22634.318,E2 22634.318} C_VEL
LIN {X 0,Y 480.881,Z 442.897,A -85,B 0,C 180,E1 22630.631,E2 22630.631} C_VEL
LIN {X 0,Y 480.887,Z 442.899,A -85,B 0,C 180,E1 22627.022,E2 22627.022} C_VEL
LIN {X 0,Y 480.955,Z 443.357,A -85,B 0,C 180,E1 22626.592,E2 22626.592} C_VEL
LIN {X 0,Y 489.811,Z 468.612,A -85,B 0,C 180,E1 22623.587,E2 22623.587} C_VEL
LIN {X 0,Y 490.976,Z 472.298,A -85,B 0,C 180,E1 22623.176,E2 22623.176} C_VEL
LIN {X 0,Y 488.386,Z 517.481,A -85,B 0,C 180,E1 22619.371,E2 22619.371} C_VEL
LIN {X 0,Y 487.345,Z 539.846,A -85,B 0,C 180,E1 22617.547,E2 22617.547} C_VEL
LIN {X 0,Y 489.365,Z 557.214,A -85,B 0,C 180,E1 22617.174,E2 22617.174} C_VEL
LIN {X 0,Y 487.59,Z 744.607,A -85,B 0,C 180,E1 22614.366,E2 22614.366} C_VEL
LIN {X 0,Y 486.997,Z 763.545,A -85,B 0,C 180,E1 22613.87,E2 22613.87} C_VEL
